    GB2312[398]:= 16#bef6;
    GB2312[399]:= 16#bff6;
    GB2312[400]:= 16#d2b1;
    GB2312[401]:= 16#c0e4;
    GB2312[402]:= 16#b6b3;
    GB2312[403]:= 16#d9fe;
    GB2312[404]:= 16#d9fd;
    GB2312[405]:= 16#bebb;
    GB2312[406]:= 16#c6e0;
    GB2312[407]:= 16#d7bc;
    GB2312[408]:= 16#daa1;
    GB2312[409]:= 16#c1b9;
    GB2312[410]:= 16#b5f2;
    GB2312[411]:= 16#c1e8;
    GB2312[412]:= 16#bcf5;
    GB2312[413]:= 16#b4d5;
    GB2312[414]:= 16#c1dd;
    GB2312[415]:= 16#c4fd;
    GB2312[416]:= 16#bcb8;
    GB2312[417]:= 16#b7b2;
    GB2312[418]:= 16#b7ef;
    GB2312[419]:= 16#d9ec;
    GB2312[420]:= 16#c6be;
    GB2312[421]:= 16#bfad;
    GB2312[422]:= 16#bbcb;
    GB2312[423]:= 16#b5ca;
    GB2312[424]:= 16#dbc9;
    GB2312[425]:= 16#d0d7;
    GB2312[426]:= 16#cdb9;
    GB2312[427]:= 16#b0bc;
    GB2312[428]:= 16#b3f6;
    GB2312[429]:= 16#bbf7;
    GB2312[430]:= 16#dbca;
    GB2312[431]:= 16#baaf;
    GB2312[432]:= 16#d4e4;
    GB2312[433]:= 16#b5b6;
    GB2312[434]:= 16#b5f3;
    GB2312[435]:= 16#d8d6;
    GB2312[436]:= 16#c8d0;
    GB2312[437]:= 16#b7d6;
    GB2312[438]:= 16#c7d0;
    GB2312[439]:= 16#d8d7;
    GB2312[440]:= 16#bfaf;
    GB2312[441]:= 16#dbbb;
    GB2312[442]:= 16#d8d8;
    GB2312[443]:= 16#d0cc;
    GB2312[444]:= 16#bbae;
    GB2312[445]:= 16#ebbe;
    GB2312[446]:= 16#c1d0;
    GB2312[447]:= 16#c1f5;
    GB2312[448]:= 16#d4f2;
    GB2312[449]:= 16#b8d5;
    GB2312[450]:= 16#b4b4;
    GB2312[451]:= 16#b3f5;
    GB2312[452]:= 16#c9be;
    GB2312[453]:= 16#c5d0;
    GB2312[454]:= 16#c5d9;
    GB2312[455]:= 16#c0fb;
    GB2312[456]:= 16#b1f0;
    GB2312[457]:= 16#d8d9;
    GB2312[458]:= 16#b9ce;
    GB2312[459]:= 16#b5bd;
    GB2312[460]:= 16#d8da;
    GB2312[461]:= 16#d6c6;
    GB2312[462]:= 16#cba2;
    GB2312[463]:= 16#c8af;
    GB2312[464]:= 16#c9b2;
    GB2312[465]:= 16#b4cc;
    GB2312[466]:= 16#bfcc;
    GB2312[467]:= 16#b9f4;
    GB2312[468]:= 16#d8db;
    GB2312[469]:= 16#d8dc;
    GB2312[470]:= 16#b6e7;
    GB2312[471]:= 16#bcc1;
    GB2312[472]:= 16#ccea;
    GB2312[473]:= 16#cff7;
    GB2312[474]:= 16#d8dd;
    GB2312[475]:= 16#c7b0;
    GB2312[476]:= 16#b9d0;
    GB2312[477]:= 16#bda3;
    GB2312[478]:= 16#ccde;
    GB2312[479]:= 16#c6ca;
    GB2312[480]:= 16#d8e0;
    GB2312[481]:= 16#d8de;
    GB2312[482]:= 16#d8df;
    GB2312[483]:= 16#b0fe;
    GB2312[484]:= 16#bee7;
    GB2312[485]:= 16#caa3;
    GB2312[486]:= 16#bcf4;
    GB2312[487]:= 16#b8b1;
    GB2312[488]:= 16#b8ee;
    GB2312[489]:= 16#d8e2;
    GB2312[490]:= 16#bdcb;
    GB2312[491]:= 16#d8e4;
    GB2312[492]:= 16#d8e3;
    GB2312[493]:= 16#c5fc;
    GB2312[494]:= 16#d8e5;
    GB2312[495]:= 16#d8e6;
    GB2312[496]:= 16#c1a6;
    GB2312[497]:= 16#c8b0;
    GB2312[498]:= 16#b0ec;
    GB2312[499]:= 16#b9a6;
    GB2312[500]:= 16#bcd3;
    GB2312[501]:= 16#cef1;
    GB2312[502]:= 16#dbbd;
    GB2312[503]:= 16#c1d3;
    GB2312[504]:= 16#b6af;
    GB2312[505]:= 16#d6fa;
    GB2312[506]:= 16#c5ac;
    GB2312[507]:= 16#bdd9;
    GB2312[508]:= 16#dbbe;
    GB2312[509]:= 16#dbbf;
    GB2312[510]:= 16#c0f8;
    GB2312[511]:= 16#bea2;
    GB2312[512]:= 16#c0cd;
    GB2312[513]:= 16#dbc0;
    GB2312[514]:= 16#cac6;
    GB2312[515]:= 16#b2aa;
    GB2312[516]:= 16#d3c2;
    GB2312[517]:= 16#c3e3;
    GB2312[518]:= 16#d1ab;
    GB2312[519]:= 16#dbc2;
    GB2312[520]:= 16#c0d5;
    GB2312[521]:= 16#dbc3;
    GB2312[522]:= 16#bfb1;
    GB2312[523]:= 16#c4bc;
    GB2312[524]:= 16#c7da;
    GB2312[525]:= 16#dbc4;
    GB2312[526]:= 16#d9e8;
    GB2312[527]:= 16#c9d7;
    GB2312[528]:= 16#b9b4;
    GB2312[529]:= 16#cef0;
    GB2312[530]:= 16#d4c8;
    GB2312[531]:= 16#b0fc;
    GB2312[532]:= 16#b4d2;
    GB2312[533]:= 16#d0d9;
    GB2312[534]:= 16#d9e9;
    GB2312[535]:= 16#decb;
    GB2312[536]:= 16#d9eb;
    GB2312[537]:= 16#d8b0;
    GB2312[538]:= 16#bbaf;
    GB2312[539]:= 16#b1b1;
    GB2312[540]:= 16#b3d7;
    GB2312[541]:= 16#d8ce;
    GB2312[542]:= 16#d4d1;
    GB2312[543]:= 16#bdb3;
    GB2312[544]:= 16#bfef;
    GB2312[545]:= 16#cfbb;
    GB2312[546]:= 16#d8d0;
    GB2312[547]:= 16#b7cb;
    GB2312[548]:= 16#d8d1;
    GB2312[549]:= 16#c6a5;
    GB2312[550]:= 16#c7f8;
    GB2312[551]:= 16#d2bd;
    GB2312[552]:= 16#d8d2;
    GB2312[553]:= 16#c4e4;
    GB2312[554]:= 16#caae;
    GB2312[555]:= 16#c7a7;
    GB2312[556]:= 16#d8a6;
    GB2312[557]:= 16#c9fd;
    GB2312[558]:= 16#cee7;
    GB2312[559]:= 16#bbdc;
    GB2312[560]:= 16#b0eb;
    GB2312[561]:= 16#bbaa;
    GB2312[562]:= 16#d0ad;
    GB2312[563]:= 16#b1b0;
    GB2312[564]:= 16#d7e4;
    GB2312[565]:= 16#d7bf;
    GB2312[566]:= 16#b5a5;
    GB2312[567]:= 16#c2f4;
    GB2312[568]:= 16#c4cf;
    GB2312[569]:= 16#b2a9;
    GB2312[570]:= 16#b2b7;
    GB2312[571]:= 16#b1e5;
    GB2312[572]:= 16#dfb2;
    GB2312[573]:= 16#d5bc;
    GB2312[574]:= 16#bfa8;
    GB2312[575]:= 16#c2ac;
    GB2312[576]:= 16#d8d5;
    GB2312[577]:= 16#c2b1;
    GB2312[578]:= 16#d8d4;
    GB2312[579]:= 16#ced4;
    GB2312[580]:= 16#dae0;
    GB2312[581]:= 16#cec0;
    GB2312[582]:= 16#d8b4;
    GB2312[583]:= 16#c3ae;
    GB2312[584]:= 16#d3a1;
    GB2312[585]:= 16#cea3;
    GB2312[586]:= 16#bcb4;
    GB2312[587]:= 16#c8b4;
    GB2312[588]:= 16#c2d1;
    GB2312[589]:= 16#beed;
    GB2312[590]:= 16#d0b6;
    GB2312[591]:= 16#dae1;
    GB2312[592]:= 16#c7e4;
    GB2312[593]:= 16#b3a7;
    GB2312[594]:= 16#b6f2;
    GB2312[595]:= 16#ccfc;
    GB2312[596]:= 16#c0fa;
    GB2312[597]:= 16#c0f7;
    GB2312[598]:= 16#d1b9;
    GB2312[599]:= 16#d1e1;
    GB2312[600]:= 16#d8c7;
    GB2312[601]:= 16#b2de;
    GB2312[602]:= 16#c0e5;
    GB2312[603]:= 16#baf1;
    GB2312[604]:= 16#d8c8;
    GB2312[605]:= 16#d4ad;
    GB2312[606]:= 16#cfe1;
    GB2312[607]:= 16#d8c9;
    GB2312[608]:= 16#d8ca;
    GB2312[609]:= 16#cfc3;
    GB2312[610]:= 16#b3f8;
    GB2312[611]:= 16#bec7;
    GB2312[612]:= 16#d8cb;
    GB2312[613]:= 16#dbcc;
    GB2312[614]:= 16#c8a5;
    GB2312[615]:= 16#cfd8;
    GB2312[616]:= 16#c8fe;
    GB2312[617]:= 16#b2ce;
    GB2312[618]:= 16#d3d6;
    GB2312[619]:= 16#b2e6;
    GB2312[620]:= 16#bcb0;
    GB2312[621]:= 16#d3d1;
    GB2312[622]:= 16#cbab;
    GB2312[623]:= 16#b7b4;
    GB2312[624]:= 16#b7a2;
    GB2312[625]:= 16#cae5;
    GB2312[626]:= 16#c8a1;
    GB2312[627]:= 16#cadc;
    GB2312[628]:= 16#b1e4;
    GB2312[629]:= 16#d0f0;
    GB2312[630]:= 16#c5d1;
    GB2312[631]:= 16#dbc5;
    GB2312[632]:= 16#b5fe;
    GB2312[633]:= 16#bfda;
    GB2312[634]:= 16#b9c5;
    GB2312[635]:= 16#bee4;
    GB2312[636]:= 16#c1ed;
    GB2312[637]:= 16#dfb6;
    GB2312[638]:= 16#dfb5;
    GB2312[639]:= 16#d6bb;
    GB2312[640]:= 16#bdd0;
    GB2312[641]:= 16#d5d9;
    GB2312[642]:= 16#b0c8;
    GB2312[643]:= 16#b6a3;
    GB2312[644]:= 16#bfc9;
    GB2312[645]:= 16#cca8;
    GB2312[646]:= 16#dfb3;
    GB2312[647]:= 16#cab7;
    GB2312[648]:= 16#d3d2;
    GB2312[649]:= 16#d8cf;
    GB2312[650]:= 16#d2b6;
    GB2312[651]:= 16#bac5;
    GB2312[652]:= 16#cbbe;
    GB2312[653]:= 16#ccbe;
    GB2312[654]:= 16#dfb7;
    GB2312[655]:= 16#b5f0;
    GB2312[656]:= 16#dfb4;
    GB2312[657]:= 16#d3f5;
    GB2312[658]:= 16#b3d4;
    GB2312[659]:= 16#b8f7;
    GB2312[660]:= 16#dfba;
    GB2312[661]:= 16#bacf;
    GB2312[662]:= 16#bcaa;
    GB2312[663]:= 16#b5f5;
    GB2312[664]:= 16#cdac;
    GB2312[665]:= 16#c3fb;
    GB2312[666]:= 16#baf3;
    GB2312[667]:= 16#c0f4;
    GB2312[668]:= 16#cdc2;
    GB2312[669]:= 16#cff2;
    GB2312[670]:= 16#dfb8;
    GB2312[671]:= 16#cfc5;
    GB2312[672]:= 16#c2c0;
    GB2312[673]:= 16#dfb9;
    GB2312[674]:= 16#c2f0;
    GB2312[675]:= 16#befd;
    GB2312[676]:= 16#c1df;
    GB2312[677]:= 16#cdcc;
    GB2312[678]:= 16#d2f7;
    GB2312[679]:= 16#b7cd;
    GB2312[680]:= 16#dfc1;
    GB2312[681]:= 16#dfc4;
    GB2312[682]:= 16#b7f1;
    GB2312[683]:= 16#b0c9;
    GB2312[684]:= 16#b6d6;
    GB2312[685]:= 16#b7d4;
    GB2312[686]:= 16#baac;
    GB2312[687]:= 16#ccfd;
    GB2312[688]:= 16#bfd4;
    GB2312[689]:= 16#cbb1;
    GB2312[690]:= 16#c6f4;
    GB2312[691]:= 16#d6a8;
    GB2312[692]:= 16#dfc5;
    GB2312[693]:= 16#cee2;
    GB2312[694]:= 16#b3b3;
    GB2312[695]:= 16#cefc;
    GB2312[696]:= 16#b4b5;
    GB2312[697]:= 16#cec7;
    GB2312[698]:= 16#baf0;
    GB2312[699]:= 16#cee1;
    GB2312[700]:= 16#d1bd;
    GB2312[701]:= 16#dfc0;
    GB2312[702]:= 16#b4f4;
    GB2312[703]:= 16#b3ca;
    GB2312[704]:= 16#b8e6;
    GB2312[705]:= 16#dfbb;
    GB2312[706]:= 16#c4c5;
    GB2312[707]:= 16#dfbc;
    GB2312[708]:= 16#dfbd;
    GB2312[709]:= 16#dfbe;
    GB2312[710]:= 16#c5bb;
    GB2312[711]:= 16#dfbf;
    GB2312[712]:= 16#dfc2;
    GB2312[713]:= 16#d4b1;
    GB2312[714]:= 16#dfc3;
    GB2312[715]:= 16#c7ba;
    GB2312[716]:= 16#ced8;
    GB2312[717]:= 16#c4d8;
    GB2312[718]:= 16#dfca;
    GB2312[719]:= 16#dfcf;
    GB2312[720]:= 16#d6dc;
    GB2312[721]:= 16#dfc9;
    GB2312[722]:= 16#dfda;
    GB2312[723]:= 16#ceb6;
    GB2312[724]:= 16#bac7;
    GB2312[725]:= 16#dfce;
    GB2312[726]:= 16#dfc8;
    GB2312[727]:= 16#c5de;
    GB2312[728]:= 16#c9eb;
    GB2312[729]:= 16#baf4;
    GB2312[730]:= 16#c3fc;
    GB2312[731]:= 16#bed7;
    GB2312[732]:= 16#dfc6;
    GB2312[733]:= 16#dfcd;
    GB2312[734]:= 16#c5d8;
    GB2312[735]:= 16#d5a6;
    GB2312[736]:= 16#bacd;
    GB2312[737]:= 16#becc;
    GB2312[738]:= 16#d3bd;
    GB2312[739]:= 16#b8c0;
    GB2312[740]:= 16#d6e4;
    GB2312[741]:= 16#dfc7;
    GB2312[742]:= 16#b9be;
    GB2312[743]:= 16#bfa7;
    GB2312[744]:= 16#c1fc;
    GB2312[745]:= 16#dfcb;
    GB2312[746]:= 16#dfcc;
    GB2312[747]:= 16#dfd0;
    GB2312[748]:= 16#dfdb;
    GB2312[749]:= 16#dfe5;
    GB2312[750]:= 16#dfd7;
    GB2312[751]:= 16#dfd6;
    GB2312[752]:= 16#d7c9;
    GB2312[753]:= 16#dfe3;
    GB2312[754]:= 16#dfe4;
    GB2312[755]:= 16#e5eb;
    GB2312[756]:= 16#d2a7;
    GB2312[757]:= 16#dfd2;
    GB2312[758]:= 16#bfa9;
    GB2312[759]:= 16#d4db;
    GB2312[760]:= 16#bfc8;
    GB2312[761]:= 16#dfd4;
    GB2312[762]:= 16#cfcc;
    GB2312[763]:= 16#dfdd;
    GB2312[764]:= 16#d1ca;
    GB2312[765]:= 16#dfde;
    GB2312[766]:= 16#b0a7;
    GB2312[767]:= 16#c6b7;
    GB2312[768]:= 16#dfd3;
    GB2312[769]:= 16#bae5;
    GB2312[770]:= 16#b6df;
    GB2312[771]:= 16#cddb;
    GB2312[772]:= 16#b9fe;
    GB2312[773]:= 16#d4d5;
    GB2312[774]:= 16#dfdf;
    GB2312[775]:= 16#cfec;
    GB2312[776]:= 16#b0a5;
    GB2312[777]:= 16#dfe7;
    GB2312[778]:= 16#dfd1;
    GB2312[779]:= 16#d1c6;
    GB2312[780]:= 16#dfd5;
    GB2312[781]:= 16#dfd8;
    GB2312[782]:= 16#dfd9;
    GB2312[783]:= 16#dfdc;
    GB2312[784]:= 16#bba9;
    GB2312[785]:= 16#dfe0;
    GB2312[786]:= 16#dfe1;
    GB2312[787]:= 16#dfe2;
    GB2312[788]:= 16#dfe6;
    GB2312[789]:= 16#dfe8;
    GB2312[790]:= 16#d3b4;
    GB2312[791]:= 16#b8e7;
    GB2312[792]:= 16#c5b6;
    GB2312[793]:= 16#dfea;
    GB2312[794]:= 16#c9da;
    GB2312[795]:= 16#c1a8;
    GB2312[796]:= 16#c4c4;
    GB2312[797]:= 16#bfde;
    GB2312[798]:= 16#cff8;
    GB2312[799]:= 16#d5dc;
    GB2312[800]:= 16#dfee;
    GB2312[801]:= 16#b2b8;
    GB2312[802]:= 16#badf;
    GB2312[803]:= 16#dfec;
    GB2312[804]:= 16#dbc1;
    GB2312[805]:= 16#d1e4;
    GB2312[806]:= 16#cbf4;
    GB2312[807]:= 16#b4bd;
    GB2312[808]:= 16#b0a6;
    GB2312[809]:= 16#dff1;
    GB2312[810]:= 16#ccc6;
    GB2312[811]:= 16#dff2;
    GB2312[812]:= 16#dfed;
    GB2312[813]:= 16#dfe9;
    GB2312[814]:= 16#dfeb;
    GB2312[815]:= 16#dfef;
    GB2312[816]:= 16#dff0;
    GB2312[817]:= 16#bbbd;
    GB2312[818]:= 16#dff3;
    GB2312[819]:= 16#dff4;
    GB2312[820]:= 16#bba3;
    GB2312[821]:= 16#cadb;
    GB2312[822]:= 16#cea8;
    GB2312[823]:= 16#e0a7;
    GB2312[824]:= 16#b3aa;
    GB2312[825]:= 16#e0a6;
    GB2312[826]:= 16#e0a1;
    GB2312[827]:= 16#dffe;
    GB2312[828]:= 16#cdd9;
    GB2312[829]:= 16#dffc;
    GB2312[830]:= 16#dffa;
    GB2312[831]:= 16#bfd0;
    GB2312[832]:= 16#d7c4;
    GB2312[833]:= 16#c9cc;
    GB2312[834]:= 16#dff8;
    GB2312[835]:= 16#b0a1;
    GB2312[836]:= 16#dffd;
    GB2312[837]:= 16#dffb;
    GB2312[838]:= 16#e0a2;
    GB2312[839]:= 16#e0a8;
    GB2312[840]:= 16#b7c8;
    GB2312[841]:= 16#c6a1;
    GB2312[842]:= 16#c9b6;
    GB2312[843]:= 16#c0b2;
    GB2312[844]:= 16#dff5;
    GB2312[845]:= 16#c5be;
    GB2312[846]:= 16#d8c4;
    GB2312[847]:= 16#dff9;
    GB2312[848]:= 16#c4f6;
    GB2312[849]:= 16#e0a3;
    GB2312[850]:= 16#e0a4;
    GB2312[851]:= 16#e0a5;
    GB2312[852]:= 16#d0a5;
    GB2312[853]:= 16#e0b4;
    GB2312[854]:= 16#cce4;
    GB2312[855]:= 16#e0b1;
    GB2312[856]:= 16#bfa6;
    GB2312[857]:= 16#e0af;
    GB2312[858]:= 16#ceb9;
    GB2312[859]:= 16#e0ab;
    GB2312[860]:= 16#c9c6;
    GB2312[861]:= 16#c0ae;
    GB2312[862]:= 16#e0ae;
    GB2312[863]:= 16#baed;
    GB2312[864]:= 16#bab0;
    GB2312[865]:= 16#e0a9;
    GB2312[866]:= 16#dff6;
    GB2312[867]:= 16#e0b3;
    GB2312[868]:= 16#e0b8;
    GB2312[869]:= 16#b4ad;
    GB2312[870]:= 16#e0b9;
    GB2312[871]:= 16#cfb2;
    GB2312[872]:= 16#bac8;
    GB2312[873]:= 16#e0b0;
    GB2312[874]:= 16#d0fa;
    GB2312[875]:= 16#e0ac;
    GB2312[876]:= 16#d4fb;
    GB2312[877]:= 16#dff7;
    GB2312[878]:= 16#c5e7;
    GB2312[879]:= 16#e0ad;
    GB2312[880]:= 16#d3f7;
    GB2312[881]:= 16#e0b6;
    GB2312[882]:= 16#e0b7;
    GB2312[883]:= 16#e0c4;
    GB2312[884]:= 16#d0e1;
    GB2312[885]:= 16#e0bc;
    GB2312[886]:= 16#e0c9;
    GB2312[887]:= 16#e0ca;
    GB2312[888]:= 16#e0be;
    GB2312[889]:= 16#e0aa;
    GB2312[890]:= 16#c9a4;
    GB2312[891]:= 16#e0c1;
    GB2312[892]:= 16#e0b2;
    GB2312[893]:= 16#cac8;
    GB2312[894]:= 16#e0c3;
    GB2312[895]:= 16#e0b5;
    GB2312[896]:= 16#cecb;
    GB2312[897]:= 16#cbc3;
    GB2312[898]:= 16#e0cd;
    GB2312[899]:= 16#e0c6;
    GB2312[900]:= 16#e0c2;
    GB2312[901]:= 16#e0cb;
    GB2312[902]:= 16#e0ba;
    GB2312[903]:= 16#e0bf;
    GB2312[904]:= 16#e0c0;
    GB2312[905]:= 16#e0c5;
    GB2312[906]:= 16#e0c7;
    GB2312[907]:= 16#e0c8;
    GB2312[908]:= 16#e0cc;
    GB2312[909]:= 16#e0bb;
    GB2312[910]:= 16#cbd4;
    GB2312[911]:= 16#e0d5;
    GB2312[912]:= 16#e0d6;
    GB2312[913]:= 16#e0d2;
    GB2312[914]:= 16#e0d0;
    GB2312[915]:= 16#bcce;
    GB2312[916]:= 16#e0d1;
    GB2312[917]:= 16#b8c2;
    GB2312[918]:= 16#d8c5;
    GB2312[919]:= 16#d0ea;
    GB2312[920]:= 16#c2ef;
    GB2312[921]:= 16#e0cf;
    GB2312[922]:= 16#e0bd;
    GB2312[923]:= 16#e0d4;
    GB2312[924]:= 16#e0d3;
    GB2312[925]:= 16#e0d7;
    GB2312[926]:= 16#e0dc;
    GB2312[927]:= 16#e0d8;
    GB2312[928]:= 16#d6f6;
    GB2312[929]:= 16#b3b0;
    GB2312[930]:= 16#d7ec;
    GB2312[931]:= 16#cbbb;
    GB2312[932]:= 16#e0da;
    GB2312[933]:= 16#cefb;
    GB2312[934]:= 16#bad9;
    GB2312[935]:= 16#e0e1;
    GB2312[936]:= 16#e0dd;
    GB2312[937]:= 16#d2ad;
    GB2312[938]:= 16#e0e2;
    GB2312[939]:= 16#e0db;
    GB2312[940]:= 16#e0d9;
    GB2312[941]:= 16#e0df;
    GB2312[942]:= 16#e0e0;
    GB2312[943]:= 16#e0de;
    GB2312[944]:= 16#e0e4;
    GB2312[945]:= 16#c6f7;
    GB2312[946]:= 16#d8ac;
    GB2312[947]:= 16#d4eb;
    GB2312[948]:= 16#e0e6;
    GB2312[949]:= 16#cac9;
    GB2312[950]:= 16#e0e5;
    GB2312[951]:= 16#b8c1;
    GB2312[952]:= 16#e0e7;
    GB2312[953]:= 16#e0e8;
    GB2312[954]:= 16#e0e9;
    GB2312[955]:= 16#e0e3;
    GB2312[956]:= 16#babf;
    GB2312[957]:= 16#cce7;
    GB2312[958]:= 16#e0ea;
    GB2312[959]:= 16#cff9;
    GB2312[960]:= 16#e0eb;
    GB2312[961]:= 16#c8c2;
    GB2312[962]:= 16#bdc0;
    GB2312[963]:= 16#c4d2;
    GB2312[964]:= 16#e0ec;
    GB2312[965]:= 16#e0ed;
    GB2312[966]:= 16#c7f4;
    GB2312[967]:= 16#cbc4;
    GB2312[968]:= 16#e0ee;
    GB2312[969]:= 16#bbd8;
    GB2312[970]:= 16#d8b6;
    GB2312[971]:= 16#d2f2;
    GB2312[972]:= 16#e0ef;
    GB2312[973]:= 16#cdc5;
    GB2312[974]:= 16#b6da;
    GB2312[975]:= 16#e0f1;
    GB2312[976]:= 16#d4b0;
    GB2312[977]:= 16#c0a7;
    GB2312[978]:= 16#b4d1;
    GB2312[979]:= 16#cea7;
    GB2312[980]:= 16#e0f0;
    GB2312[981]:= 16#e0f2;
    GB2312[982]:= 16#b9cc;
    GB2312[983]:= 16#b9fa;
    GB2312[984]:= 16#cdbc;
    GB2312[985]:= 16#e0f3;
    GB2312[986]:= 16#c6d4;
    GB2312[987]:= 16#e0f4;
    GB2312[988]:= 16#d4b2;
    GB2312[989]:= 16#c8a6;
    GB2312[990]:= 16#e0f6;
    GB2312[991]:= 16#e0f5;
    GB2312[992]:= 16#e0f7;
    GB2312[993]:= 16#cdc1;
    GB2312[994]:= 16#caa5;
    GB2312[995]:= 16#d4da;
    GB2312[996]:= 16#dbd7;
    GB2312[997]:= 16#dbd9;
    GB2312[998]:= 16#dbd8;
    GB2312[999]:= 16#b9e7;    //GB2312码 0000-999
END_IF;
(* Rung 12 *)
IF P_On THEN
    GB2312[1000]:= 16#dbdc;
    GB2312[1001]:= 16#dbdd;
    GB2312[1002]:= 16#b5d8;
    GB2312[1003]:= 16#dbda;
    GB2312[1004]:= 16#dbdb;
    GB2312[1005]:= 16#b3a1;
    GB2312[1006]:= 16#dbdf;
    GB2312[1007]:= 16#bbf8;
    GB2312[1008]:= 16#d6b7;
    GB2312[1009]:= 16#dbe0;
    GB2312[1010]:= 16#bef9;
    GB2312[1011]:= 16#b7bb;
    GB2312[1012]:= 16#dbd0;
    GB2312[1013]:= 16#ccae;
    GB2312[1014]:= 16#bfb2;
    GB2312[1015]:= 16#bbb5;
    GB2312[1016]:= 16#d7f8;
    GB2312[1017]:= 16#bfd3;
    GB2312[1018]:= 16#bfe9;
    GB2312[1019]:= 16#bce1;
    GB2312[1020]:= 16#ccb3;
    GB2312[1021]:= 16#dbde;
    GB2312[1022]:= 16#b0d3;
    GB2312[1023]:= 16#ceeb;
    GB2312[1024]:= 16#b7d8;
    GB2312[1025]:= 16#d7b9;
    GB2312[1026]:= 16#c6c2;
    GB2312[1027]:= 16#c0a4;
    GB2312[1028]:= 16#ccb9;
    GB2312[1029]:= 16#dbe7;
    GB2312[1030]:= 16#dbe1;
    GB2312[1031]:= 16#c6ba;
    GB2312[1032]:= 16#dbe3;
    GB2312[1033]:= 16#dbe8;
    GB2312[1034]:= 16#c5f7;
    GB2312[1035]:= 16#dbea;
    GB2312[1036]:= 16#dbe9;
    GB2312[1037]:= 16#bfc0;
    GB2312[1038]:= 16#dbe6;
    GB2312[1039]:= 16#dbe5;
    GB2312[1040]:= 16#b4b9;
    GB2312[1041]:= 16#c0ac;
    GB2312[1042]:= 16#c2a2;
    GB2312[1043]:= 16#dbe2;
    GB2312[1044]:= 16#dbe4;
    GB2312[1045]:= 16#d0cd;
    GB2312[1046]:= 16#dbed;
    GB2312[1047]:= 16#c0dd;
    GB2312[1048]:= 16#dbf2;
    GB2312[1049]:= 16#b6e2;
    GB2312[1050]:= 16#dbf3;
    GB2312[1051]:= 16#dbd2;
    GB2312[1052]:= 16#b9b8;
    GB2312[1053]:= 16#d4ab;
    GB2312[1054]:= 16#dbec;
    GB2312[1055]:= 16#bfd1;
    GB2312[1056]:= 16#dbf0;
    GB2312[1057]:= 16#dbd1;
    GB2312[1058]:= 16#b5e6;
    GB2312[1059]:= 16#dbeb;
    GB2312[1060]:= 16#bfe5;
    GB2312[1061]:= 16#dbee;
    GB2312[1062]:= 16#dbf1;
    GB2312[1063]:= 16#dbf9;
    GB2312[1064]:= 16#b9a1;
    GB2312[1065]:= 16#b0a3;
    GB2312[1066]:= 16#c2f1;
    GB2312[1067]:= 16#b3c7;
    GB2312[1068]:= 16#dbef;
    GB2312[1069]:= 16#dbf8;
    GB2312[1070]:= 16#c6d2;
    GB2312[1071]:= 16#dbf4;
    GB2312[1072]:= 16#dbf5;
    GB2312[1073]:= 16#dbf7;
    GB2312[1074]:= 16#dbf6;
    GB2312[1075]:= 16#dbfe;
    GB2312[1076]:= 16#d3f2;
    GB2312[1077]:= 16#b2ba;
    GB2312[1078]:= 16#dbfd;
    GB2312[1079]:= 16#dca4;
    GB2312[1080]:= 16#dbfb;
    GB2312[1081]:= 16#dbfa;
    GB2312[1082]:= 16#dbfc;
    GB2312[1083]:= 16#c5e0;
    GB2312[1084]:= 16#bbf9;
    GB2312[1085]:= 16#dca3;
    GB2312[1086]:= 16#dca5;
    GB2312[1087]:= 16#ccc3;
    GB2312[1088]:= 16#b6d1;
    GB2312[1089]:= 16#ddc0;
    GB2312[1090]:= 16#dca1;
    GB2312[1091]:= 16#dca2;
    GB2312[1092]:= 16#c7b5;
    GB2312[1093]:= 16#b6e9;
    GB2312[1094]:= 16#dca7;
    GB2312[1095]:= 16#dca6;
    GB2312[1096]:= 16#dca9;
    GB2312[1097]:= 16#b1a4;
    GB2312[1098]:= 16#b5cc;
    GB2312[1099]:= 16#bfb0;
    GB2312[1100]:= 16#d1df;
    GB2312[1101]:= 16#b6c2;
    GB2312[1102]:= 16#dca8;
    GB2312[1103]:= 16#cbfa;
    GB2312[1104]:= 16#ebf3;
    GB2312[1105]:= 16#cbdc;
    GB2312[1106]:= 16#cbfe;
    GB2312[1107]:= 16#ccc1;
    GB2312[1108]:= 16#c8fb;
    GB2312[1109]:= 16#dcaa;
    GB2312[1110]:= 16#ccee;
    GB2312[1111]:= 16#dcab;
    GB2312[1112]:= 16#dbd3;
    GB2312[1113]:= 16#dcaf;
    GB2312[1114]:= 16#dcac;
    GB2312[1115]:= 16#beb3;
    GB2312[1116]:= 16#cafb;
    GB2312[1117]:= 16#dcad;
    GB2312[1118]:= 16#c9ca;
    GB2312[1119]:= 16#c4b9;
    GB2312[1120]:= 16#c7bd;
    GB2312[1121]:= 16#dcae;
    GB2312[1122]:= 16#d4f6;
    GB2312[1123]:= 16#d0e6;
    GB2312[1124]:= 16#c4ab;
    GB2312[1125]:= 16#b6d5;
    GB2312[1126]:= 16#dbd4;
    GB2312[1127]:= 16#b1da;
    GB2312[1128]:= 16#dbd5;
    GB2312[1129]:= 16#dbd6;
    GB2312[1130]:= 16#babe;
    GB2312[1131]:= 16#c8c0;
    GB2312[1132]:= 16#cabf;
    GB2312[1133]:= 16#c8c9;
    GB2312[1134]:= 16#d7b3;
    GB2312[1135]:= 16#c9f9;
    GB2312[1136]:= 16#bfc7;
    GB2312[1137]:= 16#baf8;
    GB2312[1138]:= 16#d2bc;
    GB2312[1139]:= 16#e2ba;
    GB2312[1140]:= 16#b4a6;
    GB2312[1141]:= 16#b1b8;
    GB2312[1142]:= 16#b8b4;
    GB2312[1143]:= 16#cfc4;
    GB2312[1144]:= 16#d9e7;
    GB2312[1145]:= 16#cfa6;
    GB2312[1146]:= 16#cde2;
    GB2312[1147]:= 16#d9ed;
    GB2312[1148]:= 16#b6e0;
    GB2312[1149]:= 16#d2b9;
    GB2312[1150]:= 16#b9bb;
    GB2312[1151]:= 16#e2b9;
    GB2312[1152]:= 16#e2b7;
    GB2312[1153]:= 16#b4f3;
    GB2312[1154]:= 16#ccec;
    GB2312[1155]:= 16#ccab;
    GB2312[1156]:= 16#b7f2;
    GB2312[1157]:= 16#d8b2;
    GB2312[1158]:= 16#d1eb;
    GB2312[1159]:= 16#babb;
    GB2312[1160]:= 16#caa7;
    GB2312[1161]:= 16#cdb7;
    GB2312[1162]:= 16#d2c4;
    GB2312[1163]:= 16#bfe4;
    GB2312[1164]:= 16#bcd0;
    GB2312[1165]:= 16#b6e1;
    GB2312[1166]:= 16#dec5;
    GB2312[1167]:= 16#dec6;
    GB2312[1168]:= 16#dbbc;
    GB2312[1169]:= 16#d1d9;
    GB2312[1170]:= 16#c6e6;
    GB2312[1171]:= 16#c4ce;
    GB2312[1172]:= 16#b7ee;
    GB2312[1173]:= 16#b7dc;
    GB2312[1174]:= 16#bffc;
    GB2312[1175]:= 16#d7e0;
    GB2312[1176]:= 16#c6f5;
    GB2312[1177]:= 16#b1bc;
    GB2312[1178]:= 16#dec8;
    GB2312[1179]:= 16#bdb1;
    GB2312[1180]:= 16#ccd7;
    GB2312[1181]:= 16#deca;
    GB2312[1182]:= 16#dec9;
    GB2312[1183]:= 16#b5ec;
    GB2312[1184]:= 16#c9dd;
    GB2312[1185]:= 16#b0c2;
    GB2312[1186]:= 16#c5ae;
    GB2312[1187]:= 16#c5ab;
    GB2312[1188]:= 16#c4cc;
    GB2312[1189]:= 16#bce9;
    GB2312[1190]:= 16#cbfd;
    GB2312[1191]:= 16#bac3;
    GB2312[1192]:= 16#e5f9;
    GB2312[1193]:= 16#c8e7;
    GB2312[1194]:= 16#e5fa;
    GB2312[1195]:= 16#cdfd;
    GB2312[1196]:= 16#d7b1;
    GB2312[1197]:= 16#b8be;
    GB2312[1198]:= 16#c2e8;
    GB2312[1199]:= 16#c8d1;
    GB2312[1200]:= 16#e5fb;
    GB2312[1201]:= 16#b6ca;
    GB2312[1202]:= 16#bccb;
    GB2312[1203]:= 16#d1fd;
    GB2312[1204]:= 16#e6a1;
    GB2312[1205]:= 16#c3ee;
    GB2312[1206]:= 16#e6a4;
    GB2312[1207]:= 16#e5fe;
    GB2312[1208]:= 16#e6a5;
    GB2312[1209]:= 16#cdd7;
    GB2312[1210]:= 16#b7c1;
    GB2312[1211]:= 16#e5fc;
    GB2312[1212]:= 16#e5fd;
    GB2312[1213]:= 16#e6a3;
    GB2312[1214]:= 16#c4dd;
    GB2312[1215]:= 16#e6a8;
    GB2312[1216]:= 16#e6a7;
    GB2312[1217]:= 16#c3c3;
    GB2312[1218]:= 16#c6de;
    GB2312[1219]:= 16#e6aa;
    GB2312[1220]:= 16#c4b7;
    GB2312[1221]:= 16#e6a2;
    GB2312[1222]:= 16#cabc;
    GB2312[1223]:= 16#bde3;
    GB2312[1224]:= 16#b9c3;
    GB2312[1225]:= 16#e6a6;
    GB2312[1226]:= 16#d0d5;
    GB2312[1227]:= 16#ceaf;
    GB2312[1228]:= 16#e6a9;
    GB2312[1229]:= 16#e6b0;
    GB2312[1230]:= 16#d2a6;
    GB2312[1231]:= 16#bdaa;
    GB2312[1232]:= 16#e6ad;
    GB2312[1233]:= 16#e6af;
    GB2312[1234]:= 16#c0d1;
    GB2312[1235]:= 16#d2cc;
    GB2312[1236]:= 16#bca7;
    GB2312[1237]:= 16#e6b1;
    GB2312[1238]:= 16#d2f6;
    GB2312[1239]:= 16#d7cb;
    GB2312[1240]:= 16#cdfe;
    GB2312[1241]:= 16#cdde;
    GB2312[1242]:= 16#c2a6;
    GB2312[1243]:= 16#e6ab;
    GB2312[1244]:= 16#e6ac;
    GB2312[1245]:= 16#bdbf;
    GB2312[1246]:= 16#e6ae;
    GB2312[1247]:= 16#e6b3;
    GB2312[1248]:= 16#e6b2;
    GB2312[1249]:= 16#e6b6;
    GB2312[1250]:= 16#e6b8;
    GB2312[1251]:= 16#c4ef;
    GB2312[1252]:= 16#c4c8;
    GB2312[1253]:= 16#beea;
    GB2312[1254]:= 16#c9ef;
    GB2312[1255]:= 16#e6b7;
    GB2312[1256]:= 16#b6f0;
    GB2312[1257]:= 16#c3e4;
    GB2312[1258]:= 16#d3e9;
    GB2312[1259]:= 16#e6b4;
    GB2312[1260]:= 16#e6b5;
    GB2312[1261]:= 16#c8a2;
    GB2312[1262]:= 16#e6bd;
    GB2312[1263]:= 16#e6b9;
    GB2312[1264]:= 16#c6c5;
    GB2312[1265]:= 16#cdf1;
    GB2312[1266]:= 16#e6bb;
    GB2312[1267]:= 16#e6bc;
    GB2312[1268]:= 16#bbe9;
    GB2312[1269]:= 16#e6be;
    GB2312[1270]:= 16#e6ba;
    GB2312[1271]:= 16#c0b7;
    GB2312[1272]:= 16#d3a4;
    GB2312[1273]:= 16#e6bf;
    GB2312[1274]:= 16#c9f4;
    GB2312[1275]:= 16#e6c3;
    GB2312[1276]:= 16#e6c4;
    GB2312[1277]:= 16#d0f6;
    GB2312[1278]:= 16#c3bd;
    GB2312[1279]:= 16#c3c4;
    GB2312[1280]:= 16#e6c2;
    GB2312[1281]:= 16#e6c1;
    GB2312[1282]:= 16#e6c7;
    GB2312[1283]:= 16#cfb1;
    GB2312[1284]:= 16#ebf4;
    GB2312[1285]:= 16#e6ca;
    GB2312[1286]:= 16#e6c5;
    GB2312[1287]:= 16#bcde;
    GB2312[1288]:= 16#c9a9;
    GB2312[1289]:= 16#bcb5;
    GB2312[1290]:= 16#cfd3;
    GB2312[1291]:= 16#e6c8;
    GB2312[1292]:= 16#e6c9;
    GB2312[1293]:= 16#e6ce;
    GB2312[1294]:= 16#e6d0;
    GB2312[1295]:= 16#e6d1;
    GB2312[1296]:= 16#e6cb;
    GB2312[1297]:= 16#b5d5;
    GB2312[1298]:= 16#e6cc;
    GB2312[1299]:= 16#e6cf;
    GB2312[1300]:= 16#c4db;
    GB2312[1301]:= 16#e6c6;
    GB2312[1302]:= 16#e6cd;
    GB2312[1303]:= 16#e6d2;
    GB2312[1304]:= 16#e6d4;
    GB2312[1305]:= 16#e6d3;
    GB2312[1306]:= 16#e6d5;
    GB2312[1307]:= 16#d9f8;
    GB2312[1308]:= 16#e6d6;
    GB2312[1309]:= 16#e6d7;
    GB2312[1310]:= 16#d7d3;
    GB2312[1311]:= 16#e6dd;
    GB2312[1312]:= 16#e6de;
    GB2312[1313]:= 16#bfd7;
    GB2312[1314]:= 16#d4d0;
    GB2312[1315]:= 16#d7d6;
    GB2312[1316]:= 16#b4e6;
    GB2312[1317]:= 16#cbef;
    GB2312[1318]:= 16#e6da;
    GB2312[1319]:= 16#d8c3;
    GB2312[1320]:= 16#d7ce;
    GB2312[1321]:= 16#d0a2;
    GB2312[1322]:= 16#c3cf;
    GB2312[1323]:= 16#e6df;
    GB2312[1324]:= 16#bcbe;
    GB2312[1325]:= 16#b9c2;
    GB2312[1326]:= 16#e6db;
    GB2312[1327]:= 16#d1a7;
    GB2312[1328]:= 16#baa2;
    GB2312[1329]:= 16#c2cf;
    GB2312[1330]:= 16#d8ab;
    GB2312[1331]:= 16#caeb;
    GB2312[1332]:= 16#e5ee;
    GB2312[1333]:= 16#e6dc;
    GB2312[1334]:= 16#b7f5;
    GB2312[1335]:= 16#c8e6;
    GB2312[1336]:= 16#c4f5;
    GB2312[1337]:= 16#e5b2;
    GB2312[1338]:= 16#c4fe;
    GB2312[1339]:= 16#cbfc;
    GB2312[1340]:= 16#e5b3;
    GB2312[1341]:= 16#d5ac;
    GB2312[1342]:= 16#d3ee;
    GB2312[1343]:= 16#cad8;
    GB2312[1344]:= 16#b0b2;
    GB2312[1345]:= 16#cbce;
    GB2312[1346]:= 16#cdea;
    GB2312[1347]:= 16#baea;
    GB2312[1348]:= 16#e5b5;
    GB2312[1349]:= 16#e5b4;
    GB2312[1350]:= 16#d7da;
    GB2312[1351]:= 16#b9d9;
    GB2312[1352]:= 16#d6e6;
    GB2312[1353]:= 16#b6a8;
    GB2312[1354]:= 16#cdf0;
    GB2312[1355]:= 16#d2cb;
    GB2312[1356]:= 16#b1a6;
    GB2312[1357]:= 16#cab5;
    GB2312[1358]:= 16#b3e8;
    GB2312[1359]:= 16#c9f3;
    GB2312[1360]:= 16#bfcd;
    GB2312[1361]:= 16#d0fb;
    GB2312[1362]:= 16#cad2;
    GB2312[1363]:= 16#e5b6;
    GB2312[1364]:= 16#bbc2;
    GB2312[1365]:= 16#cfdc;
    GB2312[1366]:= 16#b9ac;
    GB2312[1367]:= 16#d4d7;
    GB2312[1368]:= 16#baa6;
    GB2312[1369]:= 16#d1e7;
    GB2312[1370]:= 16#cffc;
    GB2312[1371]:= 16#bcd2;
    GB2312[1372]:= 16#e5b7;
    GB2312[1373]:= 16#c8dd;
    GB2312[1374]:= 16#bfed;
    GB2312[1375]:= 16#b1f6;
    GB2312[1376]:= 16#cbde;
    GB2312[1377]:= 16#bcc5;
    GB2312[1378]:= 16#bcc4;
    GB2312[1379]:= 16#d2fa;
    GB2312[1380]:= 16#c3dc;
    GB2312[1381]:= 16#bfdc;
    GB2312[1382]:= 16#b8bb;
    GB2312[1383]:= 16#c3c2;
    GB2312[1384]:= 16#baae;
    GB2312[1385]:= 16#d4a2;
    GB2312[1386]:= 16#c7de;
    GB2312[1387]:= 16#c4af;
    GB2312[1388]:= 16#b2ec;
    GB2312[1389]:= 16#b9d1;
    GB2312[1390]:= 16#e5bb;
    GB2312[1391]:= 16#c1c8;
    GB2312[1392]:= 16#d5af;
    GB2312[1393]:= 16#e5bc;
    GB2312[1394]:= 16#e5be;
    GB2312[1395]:= 16#b4e7;
    GB2312[1396]:= 16#b6d4;
    GB2312[1397]:= 16#cbc2;
    GB2312[1398]:= 16#d1b0;
    GB2312[1399]:= 16#b5bc;
    GB2312[1400]:= 16#cad9;
    GB2312[1401]:= 16#b7e2;
    GB2312[1402]:= 16#c9e4;
    GB2312[1403]:= 16#bdab;
    GB2312[1404]:= 16#cebe;
    GB2312[1405]:= 16#d7f0;
    GB2312[1406]:= 16#d0a1;
    GB2312[1407]:= 16#c9d9;
    GB2312[1408]:= 16#b6fb;
    GB2312[1409]:= 16#e6d8;
    GB2312[1410]:= 16#bce2;
    GB2312[1411]:= 16#b3be;
    GB2312[1412]:= 16#c9d0;
    GB2312[1413]:= 16#e6d9;
    GB2312[1414]:= 16#b3a2;
    GB2312[1415]:= 16#decc;
    GB2312[1416]:= 16#d3c8;
    GB2312[1417]:= 16#decd;
    GB2312[1418]:= 16#d2a2;
    GB2312[1419]:= 16#dece;
    GB2312[1420]:= 16#becd;
    GB2312[1421]:= 16#decf;
    GB2312[1422]:= 16#caac;
    GB2312[1423]:= 16#d2fc;
    GB2312[1424]:= 16#b3df;
    GB2312[1425]:= 16#e5ea;
    GB2312[1426]:= 16#c4e1;
    GB2312[1427]:= 16#bea1;
    GB2312[1428]:= 16#ceb2;
    GB2312[1429]:= 16#c4f2;
    GB2312[1430]:= 16#bed6;
    GB2312[1431]:= 16#c6a8;
    GB2312[1432]:= 16#b2e3;
    GB2312[1433]:= 16#bed3;
    GB2312[1434]:= 16#c7fc;
    GB2312[1435]:= 16#cceb;
    GB2312[1436]:= 16#bdec;
    GB2312[1437]:= 16#cedd;
    GB2312[1438]:= 16#caba;
    GB2312[1439]:= 16#c6c1;
    GB2312[1440]:= 16#e5ec;
    GB2312[1441]:= 16#d0bc;
    GB2312[1442]:= 16#d5b9;
    GB2312[1443]:= 16#e5ed;
    GB2312[1444]:= 16#caf4;
    GB2312[1445]:= 16#cdc0;
    GB2312[1446]:= 16#c2c5;
    GB2312[1447]:= 16#e5ef;
    GB2312[1448]:= 16#c2c4;
    GB2312[1449]:= 16#e5f0;
    GB2312[1450]:= 16#e5f8;
    GB2312[1451]:= 16#cdcd;
    GB2312[1452]:= 16#c9bd;
    GB2312[1453]:= 16#d2d9;
    GB2312[1454]:= 16#e1a8;
    GB2312[1455]:= 16#d3ec;
    GB2312[1456]:= 16#cbea;
    GB2312[1457]:= 16#c6f1;
    GB2312[1458]:= 16#e1ac;
    GB2312[1459]:= 16#e1a7;
    GB2312[1460]:= 16#e1a9;
    GB2312[1461]:= 16#e1aa;
    GB2312[1462]:= 16#e1af;
    GB2312[1463]:= 16#b2ed;
    GB2312[1464]:= 16#e1ab;
    GB2312[1465]:= 16#b8da;
    GB2312[1466]:= 16#e1ad;
    GB2312[1467]:= 16#e1ae;
    GB2312[1468]:= 16#e1b0;
    GB2312[1469]:= 16#b5ba;
    GB2312[1470]:= 16#e1b1;
    GB2312[1471]:= 16#e1b3;
    GB2312[1472]:= 16#e1b8;
    GB2312[1473]:= 16#d1d2;
    GB2312[1474]:= 16#e1b6;
    GB2312[1475]:= 16#e1b5;
    GB2312[1476]:= 16#c1eb;
    GB2312[1477]:= 16#e1b7;
    GB2312[1478]:= 16#d4c0;
    GB2312[1479]:= 16#e1b2;
    GB2312[1480]:= 16#e1ba;
    GB2312[1481]:= 16#b0b6;
    GB2312[1482]:= 16#e1b4;
    GB2312[1483]:= 16#bff9;
    GB2312[1484]:= 16#e1b9;
    GB2312[1485]:= 16#e1bb;
    GB2312[1486]:= 16#e1be;
    GB2312[1487]:= 16#e1bc;
    GB2312[1488]:= 16#d6c5;
    GB2312[1489]:= 16#cfbf;
    GB2312[1490]:= 16#e1bd;
    GB2312[1491]:= 16#e1bf;
    GB2312[1492]:= 16#c2cd;
    GB2312[1493]:= 16#b6eb;
    GB2312[1494]:= 16#d3f8;
    GB2312[1495]:= 16#c7cd;
    GB2312[1496]:= 16#b7e5;
    GB2312[1497]:= 16#befe;
    GB2312[1498]:= 16#e1c0;
    GB2312[1499]:= 16#e1c1;
    GB2312[1500]:= 16#e1c7;
    GB2312[1501]:= 16#b3e7;
    GB2312[1502]:= 16#c6e9;
    GB2312[1503]:= 16#b4de;
    GB2312[1504]:= 16#d1c2;
    GB2312[1505]:= 16#e1c8;
    GB2312[1506]:= 16#e1c6;
    GB2312[1507]:= 16#e1c5;
    GB2312[1508]:= 16#e1c3;
    GB2312[1509]:= 16#e1c2;
    GB2312[1510]:= 16#b1c0;
    GB2312[1511]:= 16#d5b8;
    GB2312[1512]:= 16#e1c4;
    GB2312[1513]:= 16#e1cb;
    GB2312[1514]:= 16#e1cc;
    GB2312[1515]:= 16#e1ca;
    GB2312[1516]:= 16#effa;
    GB2312[1517]:= 16#e1d3;
    GB2312[1518]:= 16#e1d2;
    GB2312[1519]:= 16#c7b6;
    GB2312[1520]:= 16#e1c9;
    GB2312[1521]:= 16#e1ce;
    GB2312[1522]:= 16#e1d0;
    GB2312[1523]:= 16#e1d4;
    GB2312[1524]:= 16#e1d1;
    GB2312[1525]:= 16#e1cd;
    GB2312[1526]:= 16#e1cf;
    GB2312[1527]:= 16#e1d5;
    GB2312[1528]:= 16#e1d6;
    GB2312[1529]:= 16#e1d7;
    GB2312[1530]:= 16#e1d8;
    GB2312[1531]:= 16#e1da;
    GB2312[1532]:= 16#e1db;
    GB2312[1533]:= 16#cea1;
    GB2312[1534]:= 16#e7dd;
    GB2312[1535]:= 16#b4a8;
    GB2312[1536]:= 16#d6dd;
    GB2312[1537]:= 16#d1b2;
    GB2312[1538]:= 16#b3b2;
    GB2312[1539]:= 16#b9a4;
    GB2312[1540]:= 16#d7f3;
    GB2312[1541]:= 16#c7c9;
    GB2312[1542]:= 16#bede;
    GB2312[1543]:= 16#b9ae;
    GB2312[1544]:= 16#ced7;
    GB2312[1545]:= 16#b2ee;
    GB2312[1546]:= 16#dbcf;
    GB2312[1547]:= 16#bcba;
    GB2312[1548]:= 16#d2d1;
    GB2312[1549]:= 16#cbc8;
    GB2312[1550]:= 16#b0cd;
    GB2312[1551]:= 16#cfef;
    GB2312[1552]:= 16#d9e3;
    GB2312[1553]:= 16#bded;
    GB2312[1554]:= 16#b1d2;
    GB2312[1555]:= 16#cad0;
    GB2312[1556]:= 16#b2bc;
    GB2312[1557]:= 16#cba7;
    GB2312[1558]:= 16#b7ab;
    GB2312[1559]:= 16#caa6;
    GB2312[1560]:= 16#cfa3;
    GB2312[1561]:= 16#e0f8;
    GB2312[1562]:= 16#d5ca;
    GB2312[1563]:= 16#e0fb;
    GB2312[1564]:= 16#e0fa;
    GB2312[1565]:= 16#c5c1;
    GB2312[1566]:= 16#ccfb;
    GB2312[1567]:= 16#c1b1;
    GB2312[1568]:= 16#e0f9;
    GB2312[1569]:= 16#d6e3;
    GB2312[1570]:= 16#b2af;
    GB2312[1571]:= 16#d6c4;
    GB2312[1572]:= 16#b5db;
    GB2312[1573]:= 16#b4f8;
    GB2312[1574]:= 16#d6a1;
    GB2312[1575]:= 16#cfaf;
    GB2312[1576]:= 16#b0ef;
    GB2312[1577]:= 16#e0fc;
    GB2312[1578]:= 16#e1a1;
    GB2312[1579]:= 16#b3a3;
    GB2312[1580]:= 16#e0fd;
    GB2312[1581]:= 16#e0fe;
    GB2312[1582]:= 16#c3b1;
    GB2312[1583]:= 16#c3dd;
    GB2312[1584]:= 16#e1a2;
    GB2312[1585]:= 16#b7f9;
    GB2312[1586]:= 16#bbcf;
    GB2312[1587]:= 16#e1a3;
    GB2312[1588]:= 16#c4bb;
    GB2312[1589]:= 16#e1a4;
    GB2312[1590]:= 16#e1a5;
    GB2312[1591]:= 16#e1a6;
    GB2312[1592]:= 16#b4b1;
    GB2312[1593]:= 16#b8c9;
    GB2312[1594]:= 16#c6bd;
    GB2312[1595]:= 16#c4ea;
    GB2312[1596]:= 16#b2a2;
    GB2312[1597]:= 16#d0d2;
    GB2312[1598]:= 16#e7db;
    GB2312[1599]:= 16#bbc3;
    GB2312[1600]:= 16#d3d7;
    GB2312[1601]:= 16#d3c4;
    GB2312[1602]:= 16#b9e3;
    GB2312[1603]:= 16#e2cf;
    GB2312[1604]:= 16#d7af;
    GB2312[1605]:= 16#c7ec;
    GB2312[1606]:= 16#b1d3;
    GB2312[1607]:= 16#b4b2;
    GB2312[1608]:= 16#e2d1;
    GB2312[1609]:= 16#d0f2;
    GB2312[1610]:= 16#c2ae;
    GB2312[1611]:= 16#e2d0;
    GB2312[1612]:= 16#bfe2;
    GB2312[1613]:= 16#d3a6;
    GB2312[1614]:= 16#b5d7;
    GB2312[1615]:= 16#e2d2;
    GB2312[1616]:= 16#b5ea;
    GB2312[1617]:= 16#c3ed;
    GB2312[1618]:= 16#b8fd;
    GB2312[1619]:= 16#b8ae;
    GB2312[1620]:= 16#c5d3;
    GB2312[1621]:= 16#b7cf;
    GB2312[1622]:= 16#e2d4;
    GB2312[1623]:= 16#e2d3;
    GB2312[1624]:= 16#b6c8;
    GB2312[1625]:= 16#d7f9;
    GB2312[1626]:= 16#cda5;
    GB2312[1627]:= 16#e2d8;
    GB2312[1628]:= 16#e2d6;
    GB2312[1629]:= 16#cafc;
    GB2312[1630]:= 16#bfb5;
    GB2312[1631]:= 16#d3b9;
    GB2312[1632]:= 16#e2d5;
    GB2312[1633]:= 16#e2d7;
    GB2312[1634]:= 16#c1ae;
    GB2312[1635]:= 16#c0c8;
    GB2312[1636]:= 16#e2db;
    GB2312[1637]:= 16#e2da;
    GB2312[1638]:= 16#c0aa;
    GB2312[1639]:= 16#c1ce;
    GB2312[1640]:= 16#e2dc;
    GB2312[1641]:= 16#e2dd;
    GB2312[1642]:= 16#e2de;
    GB2312[1643]:= 16#dbc8;
    GB2312[1644]:= 16#d1d3;
    GB2312[1645]:= 16#cda2;
    GB2312[1646]:= 16#bda8;
    GB2312[1647]:= 16#dec3;
    GB2312[1648]:= 16#d8a5;
    GB2312[1649]:= 16#bfaa;
    GB2312[1650]:= 16#dbcd;
    GB2312[1651]:= 16#d2ec;
    GB2312[1652]:= 16#c6fa;
    GB2312[1653]:= 16#c5aa;
    GB2312[1654]:= 16#dec4;
    GB2312[1655]:= 16#b1d7;
    GB2312[1656]:= 16#dfae;
    GB2312[1657]:= 16#cabd;
    GB2312[1658]:= 16#dfb1;
    GB2312[1659]:= 16#b9ad;
    GB2312[1660]:= 16#d2fd;
    GB2312[1661]:= 16#b8a5;
    GB2312[1662]:= 16#baeb;
    GB2312[1663]:= 16#b3da;
    GB2312[1664]:= 16#b5dc;
    GB2312[1665]:= 16#d5c5;
    GB2312[1666]:= 16#c3d6;
    GB2312[1667]:= 16#cfd2;
    GB2312[1668]:= 16#bba1;
    GB2312[1669]:= 16#e5f3;
    GB2312[1670]:= 16#e5f2;
    GB2312[1671]:= 16#e5f4;
    GB2312[1672]:= 16#cde4;
    GB2312[1673]:= 16#c8f5;
    GB2312[1674]:= 16#b5af;
    GB2312[1675]:= 16#c7bf;
    GB2312[1676]:= 16#e5f6;
    GB2312[1677]:= 16#ecb0;
    GB2312[1678]:= 16#e5e6;
    GB2312[1679]:= 16#b9e9;
    GB2312[1680]:= 16#b5b1;
    GB2312[1681]:= 16#c2bc;
    GB2312[1682]:= 16#e5e8;
    GB2312[1683]:= 16#e5e7;
    GB2312[1684]:= 16#e5e9;
    GB2312[1685]:= 16#d2cd;
    GB2312[1686]:= 16#e1ea;
    GB2312[1687]:= 16#d0ce;
    GB2312[1688]:= 16#cdae;
    GB2312[1689]:= 16#d1e5;
    GB2312[1690]:= 16#b2ca;
    GB2312[1691]:= 16#b1eb;
    GB2312[1692]:= 16#b1f2;
    GB2312[1693]:= 16#c5ed;
    GB2312[1694]:= 16#d5c3;
    GB2312[1695]:= 16#d3b0;
    GB2312[1696]:= 16#e1dc;
    GB2312[1697]:= 16#e1dd;
    GB2312[1698]:= 16#d2db;
    GB2312[1699]:= 16#b3b9;
    GB2312[1700]:= 16#b1cb;
    GB2312[1701]:= 16#cdf9;
    GB2312[1702]:= 16#d5f7;
    GB2312[1703]:= 16#e1de;
    GB2312[1704]:= 16#beb6;
    GB2312[1705]:= 16#b4fd;
    GB2312[1706]:= 16#e1df;
    GB2312[1707]:= 16#badc;
    GB2312[1708]:= 16#e1e0;
    GB2312[1709]:= 16#bbb2;
    GB2312[1710]:= 16#c2c9;
    GB2312[1711]:= 16#e1e1;
    GB2312[1712]:= 16#d0ec;
    GB2312[1713]:= 16#cdbd;
    GB2312[1714]:= 16#e1e2;
    GB2312[1715]:= 16#b5c3;
    GB2312[1716]:= 16#c5c7;
    GB2312[1717]:= 16#e1e3;
    GB2312[1718]:= 16#e1e4;
    GB2312[1719]:= 16#d3f9;
    GB2312[1720]:= 16#e1e5;
    GB2312[1721]:= 16#d1ad;
    GB2312[1722]:= 16#e1e6;
    GB2312[1723]:= 16#cea2;
    GB2312[1724]:= 16#e1e7;
    GB2312[1725]:= 16#b5c2;
    GB2312[1726]:= 16#e1e8;
    GB2312[1727]:= 16#bbd5;
    GB2312[1728]:= 16#d0c4;
    GB2312[1729]:= 16#e2e0;
    GB2312[1730]:= 16#b1d8;
    GB2312[1731]:= 16#d2e4;
    GB2312[1732]:= 16#e2e1;
    GB2312[1733]:= 16#bcc9;
    GB2312[1734]:= 16#c8cc;
    GB2312[1735]:= 16#e2e3;
    GB2312[1736]:= 16#ecfe;
    GB2312[1737]:= 16#ecfd;
    GB2312[1738]:= 16#dfaf;
    GB2312[1739]:= 16#e2e2;
    GB2312[1740]:= 16#d6be;
    GB2312[1741]:= 16#cdfc;
    GB2312[1742]:= 16#c3a6;
    GB2312[1743]:= 16#e3c3;
    GB2312[1744]:= 16#d6d2;
    GB2312[1745]:= 16#e2e7;
    GB2312[1746]:= 16#e2e8;
    GB2312[1747]:= 16#d3c7;
    GB2312[1748]:= 16#e2ec;
    GB2312[1749]:= 16#bfec;
    GB2312[1750]:= 16#e2ed;
    GB2312[1751]:= 16#e2e5;
    GB2312[1752]:= 16#b3c0;
    GB2312[1753]:= 16#c4ee;
    GB2312[1754]:= 16#e2ee;
    GB2312[1755]:= 16#d0c3;
    GB2312[1756]:= 16#baf6;
    GB2312[1757]:= 16#e2e9;
    GB2312[1758]:= 16#b7de;
    GB2312[1759]:= 16#bbb3;
    GB2312[1760]:= 16#ccac;
    GB2312[1761]:= 16#cbcb;
    GB2312[1762]:= 16#e2e4;
    GB2312[1763]:= 16#e2e6;
    GB2312[1764]:= 16#e2ea;
    GB2312[1765]:= 16#e2eb;
    GB2312[1766]:= 16#e2f7;
    GB2312[1767]:= 16#e2f4;
    GB2312[1768]:= 16#d4f5;
    GB2312[1769]:= 16#e2f3;
    GB2312[1770]:= 16#c5ad;
    GB2312[1771]:= 16#d5fa;
    GB2312[1772]:= 16#c5c2;
    GB2312[1773]:= 16#b2c0;
    GB2312[1774]:= 16#e2ef;
    GB2312[1775]:= 16#e2f2;
    GB2312[1776]:= 16#c1af;
    GB2312[1777]:= 16#cbbc;
    GB2312[1778]:= 16#b5a1;
    GB2312[1779]:= 16#e2f9;
    GB2312[1780]:= 16#bcb1;
    GB2312[1781]:= 16#e2f1;
    GB2312[1782]:= 16#d0d4;
    GB2312[1783]:= 16#d4b9;
    GB2312[1784]:= 16#e2f5;
    GB2312[1785]:= 16#b9d6;
    GB2312[1786]:= 16#e2f6;
    GB2312[1787]:= 16#c7d3;
    GB2312[1788]:= 16#e2f0;
    GB2312[1789]:= 16#d7dc;
    GB2312[1790]:= 16#eda1;
    GB2312[1791]:= 16#e2f8;
    GB2312[1792]:= 16#eda5;
    GB2312[1793]:= 16#e2fe;
    GB2312[1794]:= 16#cad1;
    GB2312[1795]:= 16#c1b5;
    GB2312[1796]:= 16#bbd0;
    GB2312[1797]:= 16#bfd6;
    GB2312[1798]:= 16#bae3;
    GB2312[1799]:= 16#cba1;
    GB2312[1800]:= 16#eda6;
    GB2312[1801]:= 16#eda3;
    GB2312[1802]:= 16#eda2;
    GB2312[1803]:= 16#bbd6;
    GB2312[1804]:= 16#eda7;
    GB2312[1805]:= 16#d0f4;
    GB2312[1806]:= 16#eda4;
    GB2312[1807]:= 16#bade;
    GB2312[1808]:= 16#b6f7;
    GB2312[1809]:= 16#e3a1;
    GB2312[1810]:= 16#b6b2;
    GB2312[1811]:= 16#ccf1;
    GB2312[1812]:= 16#b9a7;
    GB2312[1813]:= 16#cfa2;
    GB2312[1814]:= 16#c7a1;
    GB2312[1815]:= 16#bfd2;
    GB2312[1816]:= 16#b6f1;
    GB2312[1817]:= 16#e2fa;
    GB2312[1818]:= 16#e2fb;
    GB2312[1819]:= 16#e2fd;
    GB2312[1820]:= 16#e2fc;
    GB2312[1821]:= 16#c4d5;
    GB2312[1822]:= 16#e3a2;
    GB2312[1823]:= 16#d3c1;
    GB2312[1824]:= 16#e3a7;
    GB2312[1825]:= 16#c7c4;
    GB2312[1826]:= 16#cfa4;
    GB2312[1827]:= 16#e3a9;
    GB2312[1828]:= 16#bab7;
    GB2312[1829]:= 16#e3a8;
    GB2312[1830]:= 16#bbda;
    GB2312[1831]:= 16#e3a3;
    GB2312[1832]:= 16#e3a4;
    GB2312[1833]:= 16#e3aa;
    GB2312[1834]:= 16#e3a6;
    GB2312[1835]:= 16#cef2;
    GB2312[1836]:= 16#d3c6;
    GB2312[1837]:= 16#bbbc;
    GB2312[1838]:= 16#d4c3;
    GB2312[1839]:= 16#c4fa;
    GB2312[1840]:= 16#eda8;
    GB2312[1841]:= 16#d0fc;
    GB2312[1842]:= 16#e3a5;
    GB2312[1843]:= 16#c3f5;
    GB2312[1844]:= 16#e3ad;
    GB2312[1845]:= 16#b1af;
    GB2312[1846]:= 16#e3b2;
    GB2312[1847]:= 16#bcc2;
    GB2312[1848]:= 16#e3ac;
    GB2312[1849]:= 16#b5bf;
    GB2312[1850]:= 16#c7e9;
    GB2312[1851]:= 16#e3b0;
    GB2312[1852]:= 16#beaa;
    GB2312[1853]:= 16#cdef;
    GB2312[1854]:= 16#bbf3;
    GB2312[1855]:= 16#cce8;
    GB2312[1856]:= 16#e3af;
    GB2312[1857]:= 16#e3b1;
    GB2312[1858]:= 16#cfa7;
    GB2312[1859]:= 16#e3ae;
    GB2312[1860]:= 16#cea9;
    GB2312[1861]:= 16#bbdd;
    GB2312[1862]:= 16#b5eb;
    GB2312[1863]:= 16#bee5;
    GB2312[1864]:= 16#b2d2;
    GB2312[1865]:= 16#b3cd;
    GB2312[1866]:= 16#b1b9;
    GB2312[1867]:= 16#e3ab;
    GB2312[1868]:= 16#b2d1;
    GB2312[1869]:= 16#b5ac;
    GB2312[1870]:= 16#b9df;
    GB2312[1871]:= 16#b6e8;
    GB2312[1872]:= 16#cfeb;
    GB2312[1873]:= 16#e3b7;
    GB2312[1874]:= 16#bbcc;
    GB2312[1875]:= 16#c8c7;
    GB2312[1876]:= 16#d0ca;
    GB2312[1877]:= 16#e3b8;
    GB2312[1878]:= 16#b3ee;
    GB2312[1879]:= 16#eda9;
    GB2312[1880]:= 16#d3fa;
    GB2312[1881]:= 16#d3e4;
    GB2312[1882]:= 16#edaa;
    GB2312[1883]:= 16#e3b9;
    GB2312[1884]:= 16#d2e2;
    GB2312[1885]:= 16#e3b5;
    GB2312[1886]:= 16#d3de;
    GB2312[1887]:= 16#b8d0;
    GB2312[1888]:= 16#e3b3;
    GB2312[1889]:= 16#e3b6;
    GB2312[1890]:= 16#b7df;
    GB2312[1891]:= 16#e3b4;
    GB2312[1892]:= 16#c0a2;
    GB2312[1893]:= 16#e3ba;
    GB2312[1894]:= 16#d4b8;
    GB2312[1895]:= 16#b4c8;
    GB2312[1896]:= 16#e3bb;
    GB2312[1897]:= 16#bbc5;
    GB2312[1898]:= 16#c9f7;
    GB2312[1899]:= 16#c9e5;
    GB2312[1900]:= 16#c4bd;
    GB2312[1901]:= 16#edab;
    GB2312[1902]:= 16#c2fd;
    GB2312[1903]:= 16#bbdb;
    GB2312[1904]:= 16#bfae;
    GB2312[1905]:= 16#cebf;
    GB2312[1906]:= 16#e3bc;
    GB2312[1907]:= 16#bfb6;
    GB2312[1908]:= 16#b1ef;
    GB2312[1909]:= 16#d4f7;
    GB2312[1910]:= 16#e3be;
    GB2312[1911]:= 16#edad;
    GB2312[1912]:= 16#e3bf;
    GB2312[1913]:= 16#baa9;
    GB2312[1914]:= 16#edac;
    GB2312[1915]:= 16#e3bd;
    GB2312[1916]:= 16#e3c0;
    GB2312[1917]:= 16#bab6;
    GB2312[1918]:= 16#b6ae;
    GB2312[1919]:= 16#d0b8;
    GB2312[1920]:= 16#b0c3;
    GB2312[1921]:= 16#edae;
    GB2312[1922]:= 16#edaf;
    GB2312[1923]:= 16#c0c1;
    GB2312[1924]:= 16#e3c1;
    GB2312[1925]:= 16#c5b3;
    GB2312[1926]:= 16#e3c2;
    GB2312[1927]:= 16#dcb2;
    GB2312[1928]:= 16#edb0;
    GB2312[1929]:= 16#b8ea;
    GB2312[1930]:= 16#ceec;
    GB2312[1931]:= 16#eaa7;
    GB2312[1932]:= 16#d0e7;
    GB2312[1933]:= 16#caf9;
    GB2312[1934]:= 16#c8d6;
    GB2312[1935]:= 16#cfb7;
    GB2312[1936]:= 16#b3c9;
    GB2312[1937]:= 16#ced2;
    GB2312[1938]:= 16#bde4;
    GB2312[1939]:= 16#e3de;
    GB2312[1940]:= 16#bbf2;
    GB2312[1941]:= 16#eaa8;
    GB2312[1942]:= 16#d5bd;
    GB2312[1943]:= 16#c6dd;
    GB2312[1944]:= 16#eaa9;
    GB2312[1945]:= 16#eaaa;
    GB2312[1946]:= 16#eaac;
    GB2312[1947]:= 16#eaab;
    GB2312[1948]:= 16#eaae;
    GB2312[1949]:= 16#eaad;
    GB2312[1950]:= 16#bdd8;
    GB2312[1951]:= 16#eaaf;
    GB2312[1952]:= 16#c2be;
    GB2312[1953]:= 16#b4c1;
    GB2312[1954]:= 16#b4f7;
    GB2312[1955]:= 16#bba7;
    GB2312[1956]:= 16#ece6;
    GB2312[1957]:= 16#ece5;
    GB2312[1958]:= 16#b7bf;
    GB2312[1959]:= 16#cbf9;
    GB2312[1960]:= 16#b1e2;
    GB2312[1961]:= 16#ece7;
    GB2312[1962]:= 16#c9c8;
    GB2312[1963]:= 16#ece8;
    GB2312[1964]:= 16#ece9;
    GB2312[1965]:= 16#cad6;
    GB2312[1966]:= 16#ded0;
    GB2312[1967]:= 16#b2c5;
    GB2312[1968]:= 16#d4fa;
    GB2312[1969]:= 16#c6cb;
    GB2312[1970]:= 16#b0c7;
    GB2312[1971]:= 16#b4f2;
    GB2312[1972]:= 16#c8d3;
    GB2312[1973]:= 16#cdd0;
    GB2312[1974]:= 16#bfb8;
    GB2312[1975]:= 16#bfdb;
    GB2312[1976]:= 16#c7a4;
    GB2312[1977]:= 16#d6b4;
    GB2312[1978]:= 16#c0a9;
    GB2312[1979]:= 16#ded1;
    GB2312[1980]:= 16#c9a8;
    GB2312[1981]:= 16#d1ef;
    GB2312[1982]:= 16#c5a4;
    GB2312[1983]:= 16#b0e7;
    GB2312[1984]:= 16#b3b6;
    GB2312[1985]:= 16#c8c5;
    GB2312[1986]:= 16#b0e2;
    GB2312[1987]:= 16#b7f6;
    GB2312[1988]:= 16#c5fa;
    GB2312[1989]:= 16#b6f3;
    GB2312[1990]:= 16#d5d2;
    GB2312[1991]:= 16#b3d0;
    GB2312[1992]:= 16#bcbc;
    GB2312[1993]:= 16#b3ad;
    GB2312[1994]:= 16#bef1;
    GB2312[1995]:= 16#b0d1;
    GB2312[1996]:= 16#d2d6;
    GB2312[1997]:= 16#cae3;
    GB2312[1998]:= 16#d7a5;
    GB2312[1999]:= 16#cdb6;    //GB2312码 1000-1999
END_IF;

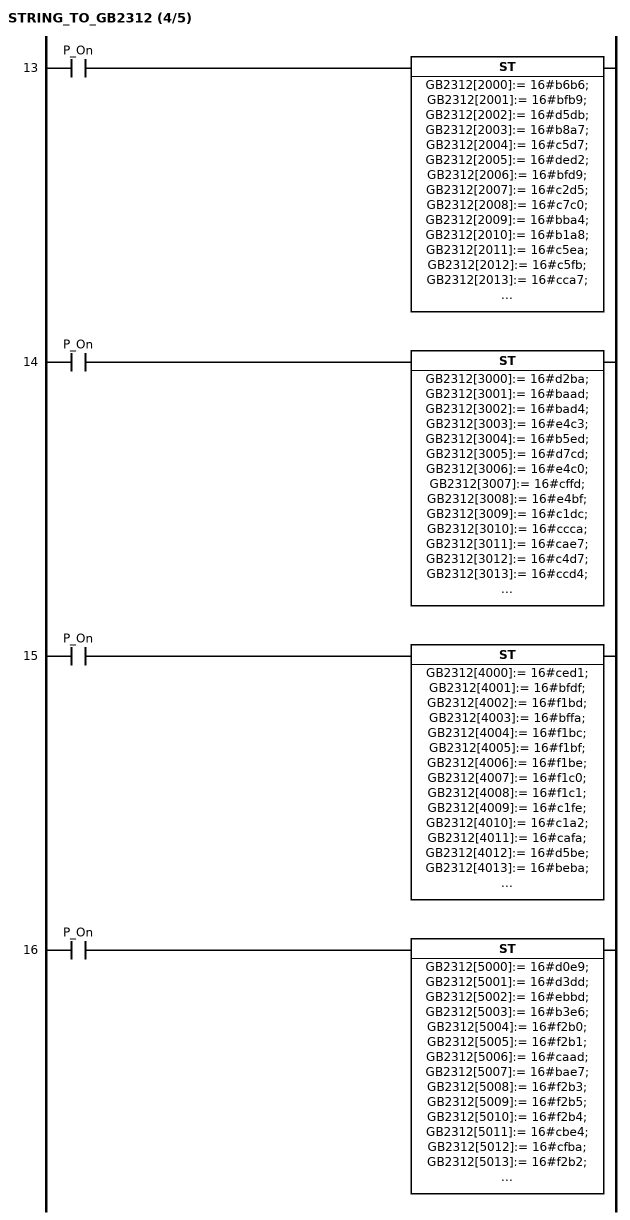
(* [picture p4: STRING_TO_GB2312, rungs 13-16] *)
(* Rung 13 *)
IF P_On THEN
    GB2312[2000]:= 16#b6b6;
    GB2312[2001]:= 16#bfb9;
    GB2312[2002]:= 16#d5db;
    GB2312[2003]:= 16#b8a7;
    GB2312[2004]:= 16#c5d7;
    GB2312[2005]:= 16#ded2;
    GB2312[2006]:= 16#bfd9;
    GB2312[2007]:= 16#c2d5;
    GB2312[2008]:= 16#c7c0;
    GB2312[2009]:= 16#bba4;
    GB2312[2010]:= 16#b1a8;
    GB2312[2011]:= 16#c5ea;
    GB2312[2012]:= 16#c5fb;
    GB2312[2013]:= 16#cca7;
    GB2312[2014]:= 16#b1a7;
    GB2312[2015]:= 16#b5d6;
    GB2312[2016]:= 16#c4a8;
    GB2312[2017]:= 16#ded3;
    GB2312[2018]:= 16#d1ba;
    GB2312[2019]:= 16#b3e9;
    GB2312[2020]:= 16#c3f2;
    GB2312[2021]:= 16#b7f7;
    GB2312[2022]:= 16#d6f4;
    GB2312[2023]:= 16#b5a3;
    GB2312[2024]:= 16#b2f0;
    GB2312[2025]:= 16#c4b4;
    GB2312[2026]:= 16#c4e9;
    GB2312[2027]:= 16#c0ad;
    GB2312[2028]:= 16#ded4;
    GB2312[2029]:= 16#b0e8;
    GB2312[2030]:= 16#c5c4;
    GB2312[2031]:= 16#c1e0;
    GB2312[2032]:= 16#b9d5;
    GB2312[2033]:= 16#bedc;
    GB2312[2034]:= 16#cdd8;
    GB2312[2035]:= 16#b0ce;
    GB2312[2036]:= 16#cdcf;
    GB2312[2037]:= 16#ded6;
    GB2312[2038]:= 16#bed0;
    GB2312[2039]:= 16#d7be;
    GB2312[2040]:= 16#ded5;
    GB2312[2041]:= 16#d5d0;
    GB2312[2042]:= 16#b0dd;
    GB2312[2043]:= 16#c4e2;
    GB2312[2044]:= 16#c2a3;
    GB2312[2045]:= 16#bcf0;
    GB2312[2046]:= 16#d3b5;
    GB2312[2047]:= 16#c0b9;
    GB2312[2048]:= 16#c5a1;
    GB2312[2049]:= 16#b2a6;
    GB2312[2050]:= 16#d4f1;
    GB2312[2051]:= 16#c0a8;
    GB2312[2052]:= 16#cac3;
    GB2312[2053]:= 16#ded7;
    GB2312[2054]:= 16#d5fc;
    GB2312[2055]:= 16#b9b0;
    GB2312[2056]:= 16#c8ad;
    GB2312[2057]:= 16#cba9;
    GB2312[2058]:= 16#ded9;
    GB2312[2059]:= 16#bfbd;
    GB2312[2060]:= 16#c6b4;
    GB2312[2061]:= 16#d7a7;
    GB2312[2062]:= 16#cab0;
    GB2312[2063]:= 16#c4c3;
    GB2312[2064]:= 16#b3d6;
    GB2312[2065]:= 16#b9d2;
    GB2312[2066]:= 16#d6b8;
    GB2312[2067]:= 16#eafc;
    GB2312[2068]:= 16#b0b4;
    GB2312[2069]:= 16#bfe6;
    GB2312[2070]:= 16#ccf4;
    GB2312[2071]:= 16#cdda;
    GB2312[2072]:= 16#d6bf;
    GB2312[2073]:= 16#c2ce;
    GB2312[2074]:= 16#cece;
    GB2312[2075]:= 16#cca2;
    GB2312[2076]:= 16#d0ae;
    GB2312[2077]:= 16#c4d3;
    GB2312[2078]:= 16#b5b2;
    GB2312[2079]:= 16#ded8;
    GB2312[2080]:= 16#d5f5;
    GB2312[2081]:= 16#bcb7;
    GB2312[2082]:= 16#bbd3;
    GB2312[2083]:= 16#b0a4;
    GB2312[2084]:= 16#c5b2;
    GB2312[2085]:= 16#b4ec;
    GB2312[2086]:= 16#d5f1;
    GB2312[2087]:= 16#eafd;
    GB2312[2088]:= 16#deda;
    GB2312[2089]:= 16#cda6;
    GB2312[2090]:= 16#cdec;
    GB2312[2091]:= 16#cee6;
    GB2312[2092]:= 16#dedc;
    GB2312[2093]:= 16#cdb1;
    GB2312[2094]:= 16#c0a6;
    GB2312[2095]:= 16#d7bd;
    GB2312[2096]:= 16#dedb;
    GB2312[2097]:= 16#b0c6;
    GB2312[2098]:= 16#bab4;
    GB2312[2099]:= 16#c9d3;
    GB2312[2100]:= 16#c4f3;
    GB2312[2101]:= 16#bee8;
    GB2312[2102]:= 16#b2b6;
    GB2312[2103]:= 16#c0cc;
    GB2312[2104]:= 16#cbf0;
    GB2312[2105]:= 16#bcf1;
    GB2312[2106]:= 16#bbbb;
    GB2312[2107]:= 16#b5b7;
    GB2312[2108]:= 16#c5f5;
    GB2312[2109]:= 16#dee6;
    GB2312[2110]:= 16#dee3;
    GB2312[2111]:= 16#bedd;
    GB2312[2112]:= 16#dedf;
    GB2312[2113]:= 16#b4b7;
    GB2312[2114]:= 16#bddd;
    GB2312[2115]:= 16#dee0;
    GB2312[2116]:= 16#c4ed;
    GB2312[2117]:= 16#cfc6;
    GB2312[2118]:= 16#b5e0;
    GB2312[2119]:= 16#b6de;
    GB2312[2120]:= 16#cada;
    GB2312[2121]:= 16#b5f4;
    GB2312[2122]:= 16#dee5;
    GB2312[2123]:= 16#d5c6;
    GB2312[2124]:= 16#dee1;
    GB2312[2125]:= 16#cccd;
    GB2312[2126]:= 16#c6fe;
    GB2312[2127]:= 16#c5c5;
    GB2312[2128]:= 16#d2b4;
    GB2312[2129]:= 16#bef2;
    GB2312[2130]:= 16#c2d3;
    GB2312[2131]:= 16#ccbd;
    GB2312[2132]:= 16#b3b8;
    GB2312[2133]:= 16#bdd3;
    GB2312[2134]:= 16#bfd8;
    GB2312[2135]:= 16#cdc6;
    GB2312[2136]:= 16#d1da;
    GB2312[2137]:= 16#b4eb;
    GB2312[2138]:= 16#dee4;
    GB2312[2139]:= 16#dedd;
    GB2312[2140]:= 16#dee7;
    GB2312[2141]:= 16#eafe;
    GB2312[2142]:= 16#c2b0;
    GB2312[2143]:= 16#dee2;
    GB2312[2144]:= 16#d6c0;
    GB2312[2145]:= 16#b5a7;
    GB2312[2146]:= 16#b2f4;
    GB2312[2147]:= 16#dee8;
    GB2312[2148]:= 16#def2;
    GB2312[2149]:= 16#deed;
    GB2312[2150]:= 16#def1;
    GB2312[2151]:= 16#c8e0;
    GB2312[2152]:= 16#d7e1;
    GB2312[2153]:= 16#deef;
    GB2312[2154]:= 16#c3e8;
    GB2312[2155]:= 16#cce1;
    GB2312[2156]:= 16#b2e5;
    GB2312[2157]:= 16#d2be;
    GB2312[2158]:= 16#deee;
    GB2312[2159]:= 16#deeb;
    GB2312[2160]:= 16#ced5;
    GB2312[2161]:= 16#b4a7;
    GB2312[2162]:= 16#bfab;
    GB2312[2163]:= 16#bebe;
    GB2312[2164]:= 16#bdd2;
    GB2312[2165]:= 16#dee9;
    GB2312[2166]:= 16#d4ae;
    GB2312[2167]:= 16#dede;
    GB2312[2168]:= 16#deea;
    GB2312[2169]:= 16#c0bf;
    GB2312[2170]:= 16#deec;
    GB2312[2171]:= 16#b2f3;
    GB2312[2172]:= 16#b8e9;
    GB2312[2173]:= 16#c2a7;
    GB2312[2174]:= 16#bdc1;
    GB2312[2175]:= 16#def5;
    GB2312[2176]:= 16#def8;
    GB2312[2177]:= 16#b2ab;
    GB2312[2178]:= 16#b4a4;
    GB2312[2179]:= 16#b4ea;
    GB2312[2180]:= 16#c9a6;
    GB2312[2181]:= 16#def6;
    GB2312[2182]:= 16#cbd1;
    GB2312[2183]:= 16#b8e3;
    GB2312[2184]:= 16#def7;
    GB2312[2185]:= 16#defa;
    GB2312[2186]:= 16#def9;
    GB2312[2187]:= 16#ccc2;
    GB2312[2188]:= 16#b0e1;
    GB2312[2189]:= 16#b4ee;
    GB2312[2190]:= 16#e5ba;
    GB2312[2191]:= 16#d0af;
    GB2312[2192]:= 16#b2eb;
    GB2312[2193]:= 16#eba1;
    GB2312[2194]:= 16#def4;
    GB2312[2195]:= 16#c9e3;
    GB2312[2196]:= 16#def3;
    GB2312[2197]:= 16#b0da;
    GB2312[2198]:= 16#d2a1;
    GB2312[2199]:= 16#b1f7;
    GB2312[2200]:= 16#ccaf;
    GB2312[2201]:= 16#def0;
    GB2312[2202]:= 16#cba4;
    GB2312[2203]:= 16#d5aa;
    GB2312[2204]:= 16#defb;
    GB2312[2205]:= 16#b4dd;
    GB2312[2206]:= 16#c4a6;
    GB2312[2207]:= 16#defd;
    GB2312[2208]:= 16#c3fe;
    GB2312[2209]:= 16#c4a1;
    GB2312[2210]:= 16#dfa1;
    GB2312[2211]:= 16#c1cc;
    GB2312[2212]:= 16#defc;
    GB2312[2213]:= 16#beef;
    GB2312[2214]:= 16#c6b2;
    GB2312[2215]:= 16#b3c5;
    GB2312[2216]:= 16#c8f6;
    GB2312[2217]:= 16#cbba;
    GB2312[2218]:= 16#defe;
    GB2312[2219]:= 16#dfa4;
    GB2312[2220]:= 16#d7b2;
    GB2312[2221]:= 16#b3b7;
    GB2312[2222]:= 16#c1c3;
    GB2312[2223]:= 16#c7cb;
    GB2312[2224]:= 16#b2a5;
    GB2312[2225]:= 16#b4e9;
    GB2312[2226]:= 16#d7ab;
    GB2312[2227]:= 16#c4ec;
    GB2312[2228]:= 16#dfa2;
    GB2312[2229]:= 16#dfa3;
    GB2312[2230]:= 16#dfa5;
    GB2312[2231]:= 16#bab3;
    GB2312[2232]:= 16#dfa6;
    GB2312[2233]:= 16#c0de;
    GB2312[2234]:= 16#c9c3;
    GB2312[2235]:= 16#b2d9;
    GB2312[2236]:= 16#c7e6;
    GB2312[2237]:= 16#dfa7;
    GB2312[2238]:= 16#c7dc;
    GB2312[2239]:= 16#dfa8;
    GB2312[2240]:= 16#eba2;
    GB2312[2241]:= 16#cbd3;
    GB2312[2242]:= 16#dfaa;
    GB2312[2243]:= 16#dfa9;
    GB2312[2244]:= 16#b2c1;
    GB2312[2245]:= 16#c5ca;
    GB2312[2246]:= 16#dfab;
    GB2312[2247]:= 16#d4dc;
    GB2312[2248]:= 16#c8c1;
    GB2312[2249]:= 16#dfac;
    GB2312[2250]:= 16#bef0;
    GB2312[2251]:= 16#dfad;
    GB2312[2252]:= 16#d6a7;
    GB2312[2253]:= 16#eab7;
    GB2312[2254]:= 16#ebb6;
    GB2312[2255]:= 16#cad5;
    GB2312[2256]:= 16#d8fc;
    GB2312[2257]:= 16#b8c4;
    GB2312[2258]:= 16#b9a5;
    GB2312[2259]:= 16#b7c5;
    GB2312[2260]:= 16#d5fe;
    GB2312[2261]:= 16#b9ca;
    GB2312[2262]:= 16#d0a7;
    GB2312[2263]:= 16#f4cd;
    GB2312[2264]:= 16#b5d0;
    GB2312[2265]:= 16#c3f4;
    GB2312[2266]:= 16#bec8;
    GB2312[2267]:= 16#ebb7;
    GB2312[2268]:= 16#b0bd;
    GB2312[2269]:= 16#bdcc;
    GB2312[2270]:= 16#c1b2;
    GB2312[2271]:= 16#b1d6;
    GB2312[2272]:= 16#b3a8;
    GB2312[2273]:= 16#b8d2;
    GB2312[2274]:= 16#c9a2;
    GB2312[2275]:= 16#b6d8;
    GB2312[2276]:= 16#ebb8;
    GB2312[2277]:= 16#beb4;
    GB2312[2278]:= 16#cafd;
    GB2312[2279]:= 16#c7c3;
    GB2312[2280]:= 16#d5fb;
    GB2312[2281]:= 16#b7f3;
    GB2312[2282]:= 16#cec4;
    GB2312[2283]:= 16#d5ab;
    GB2312[2284]:= 16#b1f3;
    GB2312[2285]:= 16#ecb3;
    GB2312[2286]:= 16#b0df;
    GB2312[2287]:= 16#ecb5;
    GB2312[2288]:= 16#b6b7;
    GB2312[2289]:= 16#c1cf;
    GB2312[2290]:= 16#f5fa;
    GB2312[2291]:= 16#d0b1;
    GB2312[2292]:= 16#d5e5;
    GB2312[2293]:= 16#ced3;
    GB2312[2294]:= 16#bdef;
    GB2312[2295]:= 16#b3e2;
    GB2312[2296]:= 16#b8ab;
    GB2312[2297]:= 16#d5b6;
    GB2312[2298]:= 16#edbd;
    GB2312[2299]:= 16#b6cf;
    GB2312[2300]:= 16#cbb9;
    GB2312[2301]:= 16#d0c2;
    GB2312[2302]:= 16#b7bd;
    GB2312[2303]:= 16#ecb6;
    GB2312[2304]:= 16#caa9;
    GB2312[2305]:= 16#c5d4;
    GB2312[2306]:= 16#ecb9;
    GB2312[2307]:= 16#ecb8;
    GB2312[2308]:= 16#c2c3;
    GB2312[2309]:= 16#ecb7;
    GB2312[2310]:= 16#d0fd;
    GB2312[2311]:= 16#ecba;
    GB2312[2312]:= 16#ecbb;
    GB2312[2313]:= 16#d7e5;
    GB2312[2314]:= 16#ecbc;
    GB2312[2315]:= 16#ecbd;
    GB2312[2316]:= 16#c6ec;
    GB2312[2317]:= 16#cede;
    GB2312[2318]:= 16#bcc8;
    GB2312[2319]:= 16#c8d5;
    GB2312[2320]:= 16#b5a9;
    GB2312[2321]:= 16#bec9;
    GB2312[2322]:= 16#d6bc;
    GB2312[2323]:= 16#d4e7;
    GB2312[2324]:= 16#d1ae;
    GB2312[2325]:= 16#d0f1;
    GB2312[2326]:= 16#eab8;
    GB2312[2327]:= 16#eab9;
    GB2312[2328]:= 16#eaba;
    GB2312[2329]:= 16#bab5;
    GB2312[2330]:= 16#cab1;
    GB2312[2331]:= 16#bff5;
    GB2312[2332]:= 16#cdfa;
    GB2312[2333]:= 16#eac0;
    GB2312[2334]:= 16#b0ba;
    GB2312[2335]:= 16#eabe;
    GB2312[2336]:= 16#c0a5;
    GB2312[2337]:= 16#eabb;
    GB2312[2338]:= 16#b2fd;
    GB2312[2339]:= 16#c3f7;
    GB2312[2340]:= 16#bbe8;
    GB2312[2341]:= 16#d2d7;
    GB2312[2342]:= 16#cef4;
    GB2312[2343]:= 16#eabf;
    GB2312[2344]:= 16#eabc;
    GB2312[2345]:= 16#eac3;
    GB2312[2346]:= 16#d0c7;
    GB2312[2347]:= 16#d3b3;
    GB2312[2348]:= 16#b4ba;
    GB2312[2349]:= 16#c3c1;
    GB2312[2350]:= 16#d7f2;
    GB2312[2351]:= 16#d5d1;
    GB2312[2352]:= 16#cac7;
    GB2312[2353]:= 16#eac5;
    GB2312[2354]:= 16#eac4;
    GB2312[2355]:= 16#eac7;
    GB2312[2356]:= 16#eac6;
    GB2312[2357]:= 16#d6e7;
    GB2312[2358]:= 16#cfd4;
    GB2312[2359]:= 16#eacb;
    GB2312[2360]:= 16#bbce;
    GB2312[2361]:= 16#bdfa;
    GB2312[2362]:= 16#c9ce;
    GB2312[2363]:= 16#eacc;
    GB2312[2364]:= 16#c9b9;
    GB2312[2365]:= 16#cffe;
    GB2312[2366]:= 16#eaca;
    GB2312[2367]:= 16#d4ce;
    GB2312[2368]:= 16#eacd;
    GB2312[2369]:= 16#eacf;
    GB2312[2370]:= 16#cded;
    GB2312[2371]:= 16#eac9;
    GB2312[2372]:= 16#eace;
    GB2312[2373]:= 16#ceee;
    GB2312[2374]:= 16#bbde;
    GB2312[2375]:= 16#b3bf;
    GB2312[2376]:= 16#c6d5;
    GB2312[2377]:= 16#beb0;
    GB2312[2378]:= 16#cefa;
    GB2312[2379]:= 16#c7e7;
    GB2312[2380]:= 16#bea7;
    GB2312[2381]:= 16#ead0;
    GB2312[2382]:= 16#d6c7;
    GB2312[2383]:= 16#c1c0;
    GB2312[2384]:= 16#d4dd;
    GB2312[2385]:= 16#ead1;
    GB2312[2386]:= 16#cfbe;
    GB2312[2387]:= 16#ead2;
    GB2312[2388]:= 16#caee;
    GB2312[2389]:= 16#c5af;
    GB2312[2390]:= 16#b0b5;
    GB2312[2391]:= 16#ead4;
    GB2312[2392]:= 16#ead3;
    GB2312[2393]:= 16#f4df;
    GB2312[2394]:= 16#c4ba;
    GB2312[2395]:= 16#b1a9;
    GB2312[2396]:= 16#e5df;
    GB2312[2397]:= 16#ead5;
    GB2312[2398]:= 16#caef;
    GB2312[2399]:= 16#ead6;
    GB2312[2400]:= 16#ead7;
    GB2312[2401]:= 16#c6d8;
    GB2312[2402]:= 16#ead8;
    GB2312[2403]:= 16#ead9;
    GB2312[2404]:= 16#d4bb;
    GB2312[2405]:= 16#c7fa;
    GB2312[2406]:= 16#d2b7;
    GB2312[2407]:= 16#b8fc;
    GB2312[2408]:= 16#eac2;
    GB2312[2409]:= 16#b2dc;
    GB2312[2410]:= 16#c2fc;
    GB2312[2411]:= 16#d4f8;
    GB2312[2412]:= 16#cce6;
    GB2312[2413]:= 16#d7ee;
    GB2312[2414]:= 16#d4c2;
    GB2312[2415]:= 16#d3d0;
    GB2312[2416]:= 16#ebc3;
    GB2312[2417]:= 16#c5f3;
    GB2312[2418]:= 16#b7fe;
    GB2312[2419]:= 16#ebd4;
    GB2312[2420]:= 16#cbb7;
    GB2312[2421]:= 16#ebde;
    GB2312[2422]:= 16#c0ca;
    GB2312[2423]:= 16#cdfb;
    GB2312[2424]:= 16#b3af;
    GB2312[2425]:= 16#c6da;
    GB2312[2426]:= 16#ebfc;
    GB2312[2427]:= 16#c4be;
    GB2312[2428]:= 16#ceb4;
    GB2312[2429]:= 16#c4a9;
    GB2312[2430]:= 16#b1be;
    GB2312[2431]:= 16#d4fd;
    GB2312[2432]:= 16#caf5;
    GB2312[2433]:= 16#d6ec;
    GB2312[2434]:= 16#c6d3;
    GB2312[2435]:= 16#b6e4;
    GB2312[2436]:= 16#bbfa;
    GB2312[2437]:= 16#d0e0;
    GB2312[2438]:= 16#c9b1;
    GB2312[2439]:= 16#d4d3;
    GB2312[2440]:= 16#c8a8;
    GB2312[2441]:= 16#b8cb;
    GB2312[2442]:= 16#e8be;
    GB2312[2443]:= 16#c9bc;
    GB2312[2444]:= 16#e8bb;
    GB2312[2445]:= 16#c0ee;
    GB2312[2446]:= 16#d0d3;
    GB2312[2447]:= 16#b2c4;
    GB2312[2448]:= 16#b4e5;
    GB2312[2449]:= 16#e8bc;
    GB2312[2450]:= 16#d5c8;
    GB2312[2451]:= 16#b6c5;
    GB2312[2452]:= 16#e8bd;
    GB2312[2453]:= 16#caf8;
    GB2312[2454]:= 16#b8dc;
    GB2312[2455]:= 16#ccf5;
    GB2312[2456]:= 16#c0b4;
    GB2312[2457]:= 16#d1ee;
    GB2312[2458]:= 16#e8bf;
    GB2312[2459]:= 16#e8c2;
    GB2312[2460]:= 16#babc;
    GB2312[2461]:= 16#b1ad;
    GB2312[2462]:= 16#bddc;
    GB2312[2463]:= 16#eabd;
    GB2312[2464]:= 16#e8c3;
    GB2312[2465]:= 16#e8c6;
    GB2312[2466]:= 16#e8cb;
    GB2312[2467]:= 16#e8cc;
    GB2312[2468]:= 16#cbc9;
    GB2312[2469]:= 16#b0e5;
    GB2312[2470]:= 16#bcab;
    GB2312[2471]:= 16#b9b9;
    GB2312[2472]:= 16#e8c1;
    GB2312[2473]:= 16#cdf7;
    GB2312[2474]:= 16#e8ca;
    GB2312[2475]:= 16#cef6;
    GB2312[2476]:= 16#d5ed;
    GB2312[2477]:= 16#c1d6;
    GB2312[2478]:= 16#e8c4;
    GB2312[2479]:= 16#c3b6;
    GB2312[2480]:= 16#b9fb;
    GB2312[2481]:= 16#d6a6;
    GB2312[2482]:= 16#e8c8;
    GB2312[2483]:= 16#cae0;
    GB2312[2484]:= 16#d4e6;
    GB2312[2485]:= 16#e8c0;
    GB2312[2486]:= 16#e8c5;
    GB2312[2487]:= 16#e8c7;
    GB2312[2488]:= 16#c7b9;
    GB2312[2489]:= 16#b7e3;
    GB2312[2490]:= 16#e8c9;
    GB2312[2491]:= 16#bfdd;
    GB2312[2492]:= 16#e8d2;
    GB2312[2493]:= 16#e8d7;
    GB2312[2494]:= 16#e8d5;
    GB2312[2495]:= 16#bcdc;
    GB2312[2496]:= 16#bccf;
    GB2312[2497]:= 16#e8db;
    GB2312[2498]:= 16#e8de;
    GB2312[2499]:= 16#e8da;
    GB2312[2500]:= 16#b1fa;
    GB2312[2501]:= 16#b0d8;
    GB2312[2502]:= 16#c4b3;
    GB2312[2503]:= 16#b8cc;
    GB2312[2504]:= 16#c6e2;
    GB2312[2505]:= 16#c8be;
    GB2312[2506]:= 16#c8e1;
    GB2312[2507]:= 16#e8cf;
    GB2312[2508]:= 16#e8d4;
    GB2312[2509]:= 16#e8d6;
    GB2312[2510]:= 16#b9f1;
    GB2312[2511]:= 16#e8d8;
    GB2312[2512]:= 16#d7f5;
    GB2312[2513]:= 16#c4fb;
    GB2312[2514]:= 16#e8dc;
    GB2312[2515]:= 16#b2e9;
    GB2312[2516]:= 16#e8d1;
    GB2312[2517]:= 16#bced;
    GB2312[2518]:= 16#bfc2;
    GB2312[2519]:= 16#e8cd;
    GB2312[2520]:= 16#d6f9;
    GB2312[2521]:= 16#c1f8;
    GB2312[2522]:= 16#b2f1;
    GB2312[2523]:= 16#e8df;
    GB2312[2524]:= 16#cac1;
    GB2312[2525]:= 16#e8d9;
    GB2312[2526]:= 16#d5a4;
    GB2312[2527]:= 16#b1ea;
    GB2312[2528]:= 16#d5bb;
    GB2312[2529]:= 16#e8ce;
    GB2312[2530]:= 16#e8d0;
    GB2312[2531]:= 16#b6b0;
    GB2312[2532]:= 16#e8d3;
    GB2312[2533]:= 16#e8dd;
    GB2312[2534]:= 16#c0b8;
    GB2312[2535]:= 16#caf7;
    GB2312[2536]:= 16#cba8;
    GB2312[2537]:= 16#c6dc;
    GB2312[2538]:= 16#c0f5;
    GB2312[2539]:= 16#e8e9;
    GB2312[2540]:= 16#d0a3;
    GB2312[2541]:= 16#e8f2;
    GB2312[2542]:= 16#d6ea;
    GB2312[2543]:= 16#e8e0;
    GB2312[2544]:= 16#e8e1;
    GB2312[2545]:= 16#d1f9;
    GB2312[2546]:= 16#bacb;
    GB2312[2547]:= 16#b8f9;
    GB2312[2548]:= 16#b8f1;
    GB2312[2549]:= 16#d4d4;
    GB2312[2550]:= 16#e8ef;
    GB2312[2551]:= 16#e8ee;
    GB2312[2552]:= 16#e8ec;
    GB2312[2553]:= 16#b9f0;
    GB2312[2554]:= 16#ccd2;
    GB2312[2555]:= 16#e8e6;
    GB2312[2556]:= 16#cea6;
    GB2312[2557]:= 16#bff2;
    GB2312[2558]:= 16#b0b8;
    GB2312[2559]:= 16#e8f1;
    GB2312[2560]:= 16#e8f0;
    GB2312[2561]:= 16#d7c0;
    GB2312[2562]:= 16#e8e4;
    GB2312[2563]:= 16#cda9;
    GB2312[2564]:= 16#c9a3;
    GB2312[2565]:= 16#bbb8;
    GB2312[2566]:= 16#bddb;
    GB2312[2567]:= 16#e8ea;
    GB2312[2568]:= 16#e8e2;
    GB2312[2569]:= 16#e8e3;
    GB2312[2570]:= 16#e8e5;
    GB2312[2571]:= 16#b5b5;
    GB2312[2572]:= 16#e8e7;
    GB2312[2573]:= 16#c7c5;
    GB2312[2574]:= 16#e8eb;
    GB2312[2575]:= 16#e8ed;
    GB2312[2576]:= 16#bdb0;
    GB2312[2577]:= 16#d7ae;
    GB2312[2578]:= 16#e8f8;
    GB2312[2579]:= 16#e8f5;
    GB2312[2580]:= 16#cdb0;
    GB2312[2581]:= 16#e8f6;
    GB2312[2582]:= 16#c1ba;
    GB2312[2583]:= 16#e8e8;
    GB2312[2584]:= 16#c3b7;
    GB2312[2585]:= 16#b0f0;
    GB2312[2586]:= 16#e8f4;
    GB2312[2587]:= 16#e8f7;
    GB2312[2588]:= 16#b9a3;
    GB2312[2589]:= 16#c9d2;
    GB2312[2590]:= 16#c3ce;
    GB2312[2591]:= 16#cee0;
    GB2312[2592]:= 16#c0e6;
    GB2312[2593]:= 16#cbf3;
    GB2312[2594]:= 16#ccdd;
    GB2312[2595]:= 16#d0b5;
    GB2312[2596]:= 16#cae1;
    GB2312[2597]:= 16#e8f3;
    GB2312[2598]:= 16#bcec;
    GB2312[2599]:= 16#e8f9;
    GB2312[2600]:= 16#c3de;
    GB2312[2601]:= 16#c6e5;
    GB2312[2602]:= 16#b9f7;
    GB2312[2603]:= 16#b0f4;
    GB2312[2604]:= 16#d7d8;
    GB2312[2605]:= 16#bcac;
    GB2312[2606]:= 16#c5ef;
    GB2312[2607]:= 16#ccc4;
    GB2312[2608]:= 16#e9a6;
    GB2312[2609]:= 16#c9ad;
    GB2312[2610]:= 16#e9a2;
    GB2312[2611]:= 16#c0e2;
    GB2312[2612]:= 16#bfc3;
    GB2312[2613]:= 16#e8fe;
    GB2312[2614]:= 16#b9d7;
    GB2312[2615]:= 16#e8fb;
    GB2312[2616]:= 16#e9a4;
    GB2312[2617]:= 16#d2ce;
    GB2312[2618]:= 16#e9a3;
    GB2312[2619]:= 16#d6b2;
    GB2312[2620]:= 16#d7b5;
    GB2312[2621]:= 16#e9a7;
    GB2312[2622]:= 16#bdb7;
    GB2312[2623]:= 16#e8fc;
    GB2312[2624]:= 16#e8fd;
    GB2312[2625]:= 16#e9a1;
    GB2312[2626]:= 16#cdd6;
    GB2312[2627]:= 16#d2ac;
    GB2312[2628]:= 16#e9b2;
    GB2312[2629]:= 16#e9a9;
    GB2312[2630]:= 16#b4aa;
    GB2312[2631]:= 16#b4bb;
    GB2312[2632]:= 16#e9ab;
    GB2312[2633]:= 16#d0a8;
    GB2312[2634]:= 16#e9a5;
    GB2312[2635]:= 16#b3fe;
    GB2312[2636]:= 16#e9ac;
    GB2312[2637]:= 16#c0e3;
    GB2312[2638]:= 16#e9aa;
    GB2312[2639]:= 16#e9b9;
    GB2312[2640]:= 16#e9b8;
    GB2312[2641]:= 16#e9ae;
    GB2312[2642]:= 16#e8fa;
    GB2312[2643]:= 16#e9a8;
    GB2312[2644]:= 16#bfac;
    GB2312[2645]:= 16#e9b1;
    GB2312[2646]:= 16#e9ba;
    GB2312[2647]:= 16#c2a5;
    GB2312[2648]:= 16#e9af;
    GB2312[2649]:= 16#b8c5;
    GB2312[2650]:= 16#e9ad;
    GB2312[2651]:= 16#d3dc;
    GB2312[2652]:= 16#e9b4;
    GB2312[2653]:= 16#e9b5;
    GB2312[2654]:= 16#e9b7;
    GB2312[2655]:= 16#e9c7;
    GB2312[2656]:= 16#c0c6;
    GB2312[2657]:= 16#e9c5;
    GB2312[2658]:= 16#e9b0;
    GB2312[2659]:= 16#e9bb;
    GB2312[2660]:= 16#b0f1;
    GB2312[2661]:= 16#e9bc;
    GB2312[2662]:= 16#d5a5;
    GB2312[2663]:= 16#e9be;
    GB2312[2664]:= 16#e9bf;
    GB2312[2665]:= 16#e9c1;
    GB2312[2666]:= 16#c1f1;
    GB2312[2667]:= 16#c8b6;
    GB2312[2668]:= 16#e9bd;
    GB2312[2669]:= 16#e9c2;
    GB2312[2670]:= 16#e9c3;
    GB2312[2671]:= 16#e9b3;
    GB2312[2672]:= 16#e9b6;
    GB2312[2673]:= 16#bbb1;
    GB2312[2674]:= 16#e9c0;
    GB2312[2675]:= 16#bcf7;
    GB2312[2676]:= 16#e9c4;
    GB2312[2677]:= 16#e9c6;
    GB2312[2678]:= 16#e9ca;
    GB2312[2679]:= 16#e9ce;
    GB2312[2680]:= 16#b2db;
    GB2312[2681]:= 16#e9c8;
    GB2312[2682]:= 16#b7ae;
    GB2312[2683]:= 16#e9cb;
    GB2312[2684]:= 16#e9cc;
    GB2312[2685]:= 16#d5c1;
    GB2312[2686]:= 16#c4a3;
    GB2312[2687]:= 16#e9d8;
    GB2312[2688]:= 16#bae1;
    GB2312[2689]:= 16#e9c9;
    GB2312[2690]:= 16#d3a3;
    GB2312[2691]:= 16#e9d4;
    GB2312[2692]:= 16#e9d7;
    GB2312[2693]:= 16#e9d0;
    GB2312[2694]:= 16#e9cf;
    GB2312[2695]:= 16#c7c1;
    GB2312[2696]:= 16#e9d2;
    GB2312[2697]:= 16#e9d9;
    GB2312[2698]:= 16#b3c8;
    GB2312[2699]:= 16#e9d3;
    GB2312[2700]:= 16#cff0;
    GB2312[2701]:= 16#e9cd;
    GB2312[2702]:= 16#b3f7;
    GB2312[2703]:= 16#e9d6;
    GB2312[2704]:= 16#e9da;
    GB2312[2705]:= 16#ccb4;
    GB2312[2706]:= 16#cfad;
    GB2312[2707]:= 16#e9d5;
    GB2312[2708]:= 16#e9dc;
    GB2312[2709]:= 16#e9db;
    GB2312[2710]:= 16#e9de;
    GB2312[2711]:= 16#e9d1;
    GB2312[2712]:= 16#e9dd;
    GB2312[2713]:= 16#e9df;
    GB2312[2714]:= 16#c3ca;
    GB2312[2715]:= 16#c7b7;
    GB2312[2716]:= 16#b4ce;
    GB2312[2717]:= 16#bbb6;
    GB2312[2718]:= 16#d0c0;
    GB2312[2719]:= 16#eca3;
    GB2312[2720]:= 16#c5b7;
    GB2312[2721]:= 16#d3fb;
    GB2312[2722]:= 16#eca4;
    GB2312[2723]:= 16#eca5;
    GB2312[2724]:= 16#c6db;
    GB2312[2725]:= 16#bfee;
    GB2312[2726]:= 16#eca6;
    GB2312[2727]:= 16#eca7;
    GB2312[2728]:= 16#d0aa;
    GB2312[2729]:= 16#c7b8;
    GB2312[2730]:= 16#b8e8;
    GB2312[2731]:= 16#eca8;
    GB2312[2732]:= 16#d6b9;
    GB2312[2733]:= 16#d5fd;
    GB2312[2734]:= 16#b4cb;
    GB2312[2735]:= 16#b2bd;
    GB2312[2736]:= 16#cee4;
    GB2312[2737]:= 16#c6e7;
    GB2312[2738]:= 16#cde1;
    GB2312[2739]:= 16#b4f5;
    GB2312[2740]:= 16#cbc0;
    GB2312[2741]:= 16#bcdf;
    GB2312[2742]:= 16#e9e2;
    GB2312[2743]:= 16#e9e3;
    GB2312[2744]:= 16#d1ea;
    GB2312[2745]:= 16#e9e5;
    GB2312[2746]:= 16#b4f9;
    GB2312[2747]:= 16#e9e4;
    GB2312[2748]:= 16#d1b3;
    GB2312[2749]:= 16#cae2;
    GB2312[2750]:= 16#b2d0;
    GB2312[2751]:= 16#e9e8;
    GB2312[2752]:= 16#e9e6;
    GB2312[2753]:= 16#e9e7;
    GB2312[2754]:= 16#d6b3;
    GB2312[2755]:= 16#e9e9;
    GB2312[2756]:= 16#e9ea;
    GB2312[2757]:= 16#e9eb;
    GB2312[2758]:= 16#e9ec;
    GB2312[2759]:= 16#ecaf;
    GB2312[2760]:= 16#c5b9;
    GB2312[2761]:= 16#b6ce;
    GB2312[2762]:= 16#d2f3;
    GB2312[2763]:= 16#b5ee;
    GB2312[2764]:= 16#bbd9;
    GB2312[2765]:= 16#ecb1;
    GB2312[2766]:= 16#d2e3;
    GB2312[2767]:= 16#cee3;
    GB2312[2768]:= 16#c4b8;
    GB2312[2769]:= 16#c3bf;
    GB2312[2770]:= 16#b6be;
    GB2312[2771]:= 16#d8b9;
    GB2312[2772]:= 16#b1c8;
    GB2312[2773]:= 16#b1cf;
    GB2312[2774]:= 16#b1d1;
    GB2312[2775]:= 16#c5fe;
    GB2312[2776]:= 16#b1d0;
    GB2312[2777]:= 16#c3ab;
    GB2312[2778]:= 16#d5b1;
    GB2312[2779]:= 16#eba4;
    GB2312[2780]:= 16#bac1;
    GB2312[2781]:= 16#ccba;
    GB2312[2782]:= 16#eba5;
    GB2312[2783]:= 16#eba7;
    GB2312[2784]:= 16#eba8;
    GB2312[2785]:= 16#eba6;
    GB2312[2786]:= 16#eba9;
    GB2312[2787]:= 16#ebab;
    GB2312[2788]:= 16#ebaa;
    GB2312[2789]:= 16#ebac;
    GB2312[2790]:= 16#cacf;
    GB2312[2791]:= 16#d8b5;
    GB2312[2792]:= 16#c3f1;
    GB2312[2793]:= 16#c3a5;
    GB2312[2794]:= 16#c6f8;
    GB2312[2795]:= 16#ebad;
    GB2312[2796]:= 16#c4ca;
    GB2312[2797]:= 16#ebae;
    GB2312[2798]:= 16#ebaf;
    GB2312[2799]:= 16#ebb0;
    GB2312[2800]:= 16#b7d5;
    GB2312[2801]:= 16#b7fa;
    GB2312[2802]:= 16#ebb1;
    GB2312[2803]:= 16#c7e2;
    GB2312[2804]:= 16#ebb3;
    GB2312[2805]:= 16#baa4;
    GB2312[2806]:= 16#d1f5;
    GB2312[2807]:= 16#b0b1;
    GB2312[2808]:= 16#ebb2;
    GB2312[2809]:= 16#ebb4;
    GB2312[2810]:= 16#b5aa;
    GB2312[2811]:= 16#c2c8;
    GB2312[2812]:= 16#c7e8;
    GB2312[2813]:= 16#ebb5;
    GB2312[2814]:= 16#cbae;
    GB2312[2815]:= 16#e3df;
    GB2312[2816]:= 16#d3c0;
    GB2312[2817]:= 16#d9db;
    GB2312[2818]:= 16#cda1;
    GB2312[2819]:= 16#d6ad;
    GB2312[2820]:= 16#c7f3;
    GB2312[2821]:= 16#d9e0;
    GB2312[2822]:= 16#bbe3;
    GB2312[2823]:= 16#baba;
    GB2312[2824]:= 16#e3e2;
    GB2312[2825]:= 16#cfab;
    GB2312[2826]:= 16#e3e0;
    GB2312[2827]:= 16#c9c7;
    GB2312[2828]:= 16#bab9;
    GB2312[2829]:= 16#d1b4;
    GB2312[2830]:= 16#e3e1;
    GB2312[2831]:= 16#c8ea;
    GB2312[2832]:= 16#b9af;
    GB2312[2833]:= 16#bdad;
    GB2312[2834]:= 16#b3d8;
    GB2312[2835]:= 16#cedb;
    GB2312[2836]:= 16#ccc0;
    GB2312[2837]:= 16#e3e8;
    GB2312[2838]:= 16#e3e9;
    GB2312[2839]:= 16#cdf4;
    GB2312[2840]:= 16#ccad;
    GB2312[2841]:= 16#bcb3;
    GB2312[2842]:= 16#e3ea;
    GB2312[2843]:= 16#e3eb;
    GB2312[2844]:= 16#d0da;
    GB2312[2845]:= 16#c6fb;
    GB2312[2846]:= 16#b7da;
    GB2312[2847]:= 16#c7df;
    GB2312[2848]:= 16#d2ca;
    GB2312[2849]:= 16#ced6;
    GB2312[2850]:= 16#e3e4;
    GB2312[2851]:= 16#e3ec;
    GB2312[2852]:= 16#c9f2;
    GB2312[2853]:= 16#b3c1;
    GB2312[2854]:= 16#e3e7;
    GB2312[2855]:= 16#c6e3;
    GB2312[2856]:= 16#e3e5;
    GB2312[2857]:= 16#edb3;
    GB2312[2858]:= 16#e3e6;
    GB2312[2859]:= 16#c9b3;
    GB2312[2860]:= 16#c5e6;
    GB2312[2861]:= 16#b9b5;
    GB2312[2862]:= 16#c3bb;
    GB2312[2863]:= 16#e3e3;
    GB2312[2864]:= 16#c5bd;
    GB2312[2865]:= 16#c1a4;
    GB2312[2866]:= 16#c2d9;
    GB2312[2867]:= 16#b2d7;
    GB2312[2868]:= 16#e3ed;
    GB2312[2869]:= 16#bba6;
    GB2312[2870]:= 16#c4ad;
    GB2312[2871]:= 16#e3f0;
    GB2312[2872]:= 16#beda;
    GB2312[2873]:= 16#e3fb;
    GB2312[2874]:= 16#e3f5;
    GB2312[2875]:= 16#bad3;
    GB2312[2876]:= 16#b7d0;
    GB2312[2877]:= 16#d3cd;
    GB2312[2878]:= 16#d6ce;
    GB2312[2879]:= 16#d5d3;
    GB2312[2880]:= 16#b9c1;
    GB2312[2881]:= 16#d5b4;
    GB2312[2882]:= 16#d1d8;
    GB2312[2883]:= 16#d0b9;
    GB2312[2884]:= 16#c7f6;
    GB2312[2885]:= 16#c8aa;
    GB2312[2886]:= 16#b2b4;
    GB2312[2887]:= 16#c3da;
    GB2312[2888]:= 16#e3ee;
    GB2312[2889]:= 16#e3fc;
    GB2312[2890]:= 16#e3ef;
    GB2312[2891]:= 16#b7a8;
    GB2312[2892]:= 16#e3f7;
    GB2312[2893]:= 16#e3f4;
    GB2312[2894]:= 16#b7ba;
    GB2312[2895]:= 16#c5a2;
    GB2312[2896]:= 16#e3f6;
    GB2312[2897]:= 16#c5dd;
    GB2312[2898]:= 16#b2a8;
    GB2312[2899]:= 16#c6fc;
    GB2312[2900]:= 16#c4e0;
    GB2312[2901]:= 16#d7a2;
    GB2312[2902]:= 16#c0e1;
    GB2312[2903]:= 16#e3f9;
    GB2312[2904]:= 16#e3fa;
    GB2312[2905]:= 16#e3fd;
    GB2312[2906]:= 16#cca9;
    GB2312[2907]:= 16#e3f3;
    GB2312[2908]:= 16#d3be;
    GB2312[2909]:= 16#b1c3;
    GB2312[2910]:= 16#edb4;
    GB2312[2911]:= 16#e3f1;
    GB2312[2912]:= 16#e3f2;
    GB2312[2913]:= 16#e3f8;
    GB2312[2914]:= 16#d0ba;
    GB2312[2915]:= 16#c6c3;
    GB2312[2916]:= 16#d4f3;
    GB2312[2917]:= 16#e3fe;
    GB2312[2918]:= 16#bde0;
    GB2312[2919]:= 16#e4a7;
    GB2312[2920]:= 16#e4a6;
    GB2312[2921]:= 16#d1f3;
    GB2312[2922]:= 16#e4a3;
    GB2312[2923]:= 16#e4a9;
    GB2312[2924]:= 16#c8f7;
    GB2312[2925]:= 16#cfb4;
    GB2312[2926]:= 16#e4a8;
    GB2312[2927]:= 16#e4ae;
    GB2312[2928]:= 16#c2e5;
    GB2312[2929]:= 16#b6b4;
    GB2312[2930]:= 16#bdf2;
    GB2312[2931]:= 16#e4a2;
    GB2312[2932]:= 16#bae9;
    GB2312[2933]:= 16#e4aa;
    GB2312[2934]:= 16#e4ac;
    GB2312[2935]:= 16#b6fd;
    GB2312[2936]:= 16#d6de;
    GB2312[2937]:= 16#e4b2;
    GB2312[2938]:= 16#e4ad;
    GB2312[2939]:= 16#e4a1;
    GB2312[2940]:= 16#bbee;
    GB2312[2941]:= 16#cddd;
    GB2312[2942]:= 16#c7a2;
    GB2312[2943]:= 16#c5c9;
    GB2312[2944]:= 16#c1f7;
    GB2312[2945]:= 16#e4a4;
    GB2312[2946]:= 16#c7b3;
    GB2312[2947]:= 16#bdac;
    GB2312[2948]:= 16#bdbd;
    GB2312[2949]:= 16#e4a5;
    GB2312[2950]:= 16#d7c7;
    GB2312[2951]:= 16#b2e2;
    GB2312[2952]:= 16#e4ab;
    GB2312[2953]:= 16#bcc3;
    GB2312[2954]:= 16#e4af;
    GB2312[2955]:= 16#bbeb;
    GB2312[2956]:= 16#e4b0;
    GB2312[2957]:= 16#c5a8;
    GB2312[2958]:= 16#e4b1;
    GB2312[2959]:= 16#d5e3;
    GB2312[2960]:= 16#bfa3;
    GB2312[2961]:= 16#e4ba;
    GB2312[2962]:= 16#e4b7;
    GB2312[2963]:= 16#e4bb;
    GB2312[2964]:= 16#e4bd;
    GB2312[2965]:= 16#c6d6;
    GB2312[2966]:= 16#bac6;
    GB2312[2967]:= 16#c0cb;
    GB2312[2968]:= 16#b8a1;
    GB2312[2969]:= 16#e4b4;
    GB2312[2970]:= 16#d4a1;
    GB2312[2971]:= 16#baa3;
    GB2312[2972]:= 16#bdfe;
    GB2312[2973]:= 16#e4bc;
    GB2312[2974]:= 16#cdbf;
    GB2312[2975]:= 16#c4f9;
    GB2312[2976]:= 16#cffb;
    GB2312[2977]:= 16#c9e6;
    GB2312[2978]:= 16#d3bf;
    GB2312[2979]:= 16#cfd1;
    GB2312[2980]:= 16#e4b3;
    GB2312[2981]:= 16#e4b8;
    GB2312[2982]:= 16#e4b9;
    GB2312[2983]:= 16#cce9;
    GB2312[2984]:= 16#ccce;
    GB2312[2985]:= 16#c0d4;
    GB2312[2986]:= 16#e4b5;
    GB2312[2987]:= 16#c1b0;
    GB2312[2988]:= 16#e4b6;
    GB2312[2989]:= 16#ced0;
    GB2312[2990]:= 16#bbc1;
    GB2312[2991]:= 16#b5d3;
    GB2312[2992]:= 16#c8f3;
    GB2312[2993]:= 16#bda7;
    GB2312[2994]:= 16#d5c7;
    GB2312[2995]:= 16#c9ac;
    GB2312[2996]:= 16#b8a2;
    GB2312[2997]:= 16#e4ca;
    GB2312[2998]:= 16#e4cc;
    GB2312[2999]:= 16#d1c4;     //GB2312码 2000-2999
END_IF;
(* Rung 14 *)
IF P_On THEN
    GB2312[3000]:= 16#d2ba;
    GB2312[3001]:= 16#baad;
    GB2312[3002]:= 16#bad4;
    GB2312[3003]:= 16#e4c3;
    GB2312[3004]:= 16#b5ed;
    GB2312[3005]:= 16#d7cd;
    GB2312[3006]:= 16#e4c0;
    GB2312[3007]:= 16#cffd;
    GB2312[3008]:= 16#e4bf;
    GB2312[3009]:= 16#c1dc;
    GB2312[3010]:= 16#ccca;
    GB2312[3011]:= 16#cae7;
    GB2312[3012]:= 16#c4d7;
    GB2312[3013]:= 16#ccd4;
    GB2312[3014]:= 16#e4c8;
    GB2312[3015]:= 16#e4c7;
    GB2312[3016]:= 16#e4c1;
    GB2312[3017]:= 16#e4c4;
    GB2312[3018]:= 16#b5ad;
    GB2312[3019]:= 16#d3d9;
    GB2312[3020]:= 16#e4c6;
    GB2312[3021]:= 16#d2f9;
    GB2312[3022]:= 16#b4e3;
    GB2312[3023]:= 16#bbb4;
    GB2312[3024]:= 16#c9ee;
    GB2312[3025]:= 16#b4be;
    GB2312[3026]:= 16#bbec;
    GB2312[3027]:= 16#d1cd;
    GB2312[3028]:= 16#cced;
    GB2312[3029]:= 16#edb5;
    GB2312[3030]:= 16#c7e5;
    GB2312[3031]:= 16#d4a8;
    GB2312[3032]:= 16#e4cb;
    GB2312[3033]:= 16#d7d5;
    GB2312[3034]:= 16#e4c2;
    GB2312[3035]:= 16#bda5;
    GB2312[3036]:= 16#e4c5;
    GB2312[3037]:= 16#d3e6;
    GB2312[3038]:= 16#e4c9;
    GB2312[3039]:= 16#c9f8;
    GB2312[3040]:= 16#e4be;
    GB2312[3041]:= 16#d3e5;
    GB2312[3042]:= 16#c7fe;
    GB2312[3043]:= 16#b6c9;
    GB2312[3044]:= 16#d4fc;
    GB2312[3045]:= 16#b2b3;
    GB2312[3046]:= 16#e4d7;
    GB2312[3047]:= 16#cec2;
    GB2312[3048]:= 16#e4cd;
    GB2312[3049]:= 16#cebc;
    GB2312[3050]:= 16#b8db;
    GB2312[3051]:= 16#e4d6;
    GB2312[3052]:= 16#bfca;
    GB2312[3053]:= 16#d3ce;
    GB2312[3054]:= 16#c3ec;
    GB2312[3055]:= 16#c5c8;
    GB2312[3056]:= 16#e4d8;
    GB2312[3057]:= 16#cdc4;
    GB2312[3058]:= 16#e4cf;
    GB2312[3059]:= 16#e4d4;
    GB2312[3060]:= 16#e4d5;
    GB2312[3061]:= 16#bafe;
    GB2312[3062]:= 16#cfe6;
    GB2312[3063]:= 16#d5bf;
    GB2312[3064]:= 16#e4d2;
    GB2312[3065]:= 16#e4d0;
    GB2312[3066]:= 16#e4ce;
    GB2312[3067]:= 16#cde5;
    GB2312[3068]:= 16#caaa;
    GB2312[3069]:= 16#c0a3;
    GB2312[3070]:= 16#bda6;
    GB2312[3071]:= 16#e4d3;
    GB2312[3072]:= 16#b8c8;
    GB2312[3073]:= 16#e4e7;
    GB2312[3074]:= 16#d4b4;
    GB2312[3075]:= 16#e4db;
    GB2312[3076]:= 16#c1ef;
    GB2312[3077]:= 16#e4e9;
    GB2312[3078]:= 16#d2e7;
    GB2312[3079]:= 16#e4df;
    GB2312[3080]:= 16#e4e0;
    GB2312[3081]:= 16#cfaa;
    GB2312[3082]:= 16#cbdd;
    GB2312[3083]:= 16#e4da;
    GB2312[3084]:= 16#e4d1;
    GB2312[3085]:= 16#e4e5;
    GB2312[3086]:= 16#c8dc;
    GB2312[3087]:= 16#e4e3;
    GB2312[3088]:= 16#c4e7;
    GB2312[3089]:= 16#e4e2;
    GB2312[3090]:= 16#e4e1;
    GB2312[3091]:= 16#b3fc;
    GB2312[3092]:= 16#e4e8;
    GB2312[3093]:= 16#b5e1;
    GB2312[3094]:= 16#d7cc;
    GB2312[3095]:= 16#e4e6;
    GB2312[3096]:= 16#bbac;
    GB2312[3097]:= 16#d7d2;
    GB2312[3098]:= 16#cccf;
    GB2312[3099]:= 16#ebf8;
    GB2312[3100]:= 16#e4e4;
    GB2312[3101]:= 16#b9f6;
    GB2312[3102]:= 16#d6cd;
    GB2312[3103]:= 16#e4d9;
    GB2312[3104]:= 16#e4dc;
    GB2312[3105]:= 16#c2fa;
    GB2312[3106]:= 16#e4de;
    GB2312[3107]:= 16#c2cb;
    GB2312[3108]:= 16#c0c4;
    GB2312[3109]:= 16#c2d0;
    GB2312[3110]:= 16#b1f5;
    GB2312[3111]:= 16#ccb2;
    GB2312[3112]:= 16#b5ce;
    GB2312[3113]:= 16#e4ef;
    GB2312[3114]:= 16#c6af;
    GB2312[3115]:= 16#c6e1;
    GB2312[3116]:= 16#e4f5;
    GB2312[3117]:= 16#c2a9;
    GB2312[3118]:= 16#c0ec;
    GB2312[3119]:= 16#d1dd;
    GB2312[3120]:= 16#e4ee;
    GB2312[3121]:= 16#c4ae;
    GB2312[3122]:= 16#e4ed;
    GB2312[3123]:= 16#e4f6;
    GB2312[3124]:= 16#e4f4;
    GB2312[3125]:= 16#c2fe;
    GB2312[3126]:= 16#e4dd;
    GB2312[3127]:= 16#e4f0;
    GB2312[3128]:= 16#cafe;
    GB2312[3129]:= 16#d5c4;
    GB2312[3130]:= 16#e4f1;
    GB2312[3131]:= 16#d1fa;
    GB2312[3132]:= 16#e4eb;
    GB2312[3133]:= 16#e4ec;
    GB2312[3134]:= 16#e4f2;
    GB2312[3135]:= 16#ceab;
    GB2312[3136]:= 16#c5cb;
    GB2312[3137]:= 16#c7b1;
    GB2312[3138]:= 16#c2ba;
    GB2312[3139]:= 16#e4ea;
    GB2312[3140]:= 16#c1ca;
    GB2312[3141]:= 16#ccb6;
    GB2312[3142]:= 16#b3b1;
    GB2312[3143]:= 16#e4fb;
    GB2312[3144]:= 16#e4f3;
    GB2312[3145]:= 16#e4fa;
    GB2312[3146]:= 16#e4fd;
    GB2312[3147]:= 16#e4fc;
    GB2312[3148]:= 16#b3ce;
    GB2312[3149]:= 16#b3ba;
    GB2312[3150]:= 16#e4f7;
    GB2312[3151]:= 16#e4f9;
    GB2312[3152]:= 16#e4f8;
    GB2312[3153]:= 16#c5ec;
    GB2312[3154]:= 16#c0bd;
    GB2312[3155]:= 16#d4e8;
    GB2312[3156]:= 16#e5a2;
    GB2312[3157]:= 16#b0c4;
    GB2312[3158]:= 16#e5a4;
    GB2312[3159]:= 16#e5a3;
    GB2312[3160]:= 16#bca4;
    GB2312[3161]:= 16#e5a5;
    GB2312[3162]:= 16#e5a1;
    GB2312[3163]:= 16#e4fe;
    GB2312[3164]:= 16#b1f4;
    GB2312[3165]:= 16#e5a8;
    GB2312[3166]:= 16#e5a9;
    GB2312[3167]:= 16#e5a6;
    GB2312[3168]:= 16#e5a7;
    GB2312[3169]:= 16#e5aa;
    GB2312[3170]:= 16#c6d9;
    GB2312[3171]:= 16#e5ab;
    GB2312[3172]:= 16#e5ad;
    GB2312[3173]:= 16#e5ac;
    GB2312[3174]:= 16#e5af;
    GB2312[3175]:= 16#e5ae;
    GB2312[3176]:= 16#b9e0;
    GB2312[3177]:= 16#e5b0;
    GB2312[3178]:= 16#e5b1;
    GB2312[3179]:= 16#bbf0;
    GB2312[3180]:= 16#ece1;
    GB2312[3181]:= 16#c3f0;
    GB2312[3182]:= 16#b5c6;
    GB2312[3183]:= 16#bbd2;
    GB2312[3184]:= 16#c1e9;
    GB2312[3185]:= 16#d4ee;
    GB2312[3186]:= 16#bec4;
    GB2312[3187]:= 16#d7c6;
    GB2312[3188]:= 16#d4d6;
    GB2312[3189]:= 16#b2d3;
    GB2312[3190]:= 16#ecbe;
    GB2312[3191]:= 16#eac1;
    GB2312[3192]:= 16#c2af;
    GB2312[3193]:= 16#b4b6;
    GB2312[3194]:= 16#d1d7;
    GB2312[3195]:= 16#b3b4;
    GB2312[3196]:= 16#c8b2;
    GB2312[3197]:= 16#bfbb;
    GB2312[3198]:= 16#ecc0;
    GB2312[3199]:= 16#d6cb;
    GB2312[3200]:= 16#ecbf;
    GB2312[3201]:= 16#ecc1;
    GB2312[3202]:= 16#ecc5;
    GB2312[3203]:= 16#bee6;
    GB2312[3204]:= 16#ccbf;
    GB2312[3205]:= 16#c5da;
    GB2312[3206]:= 16#bebc;
    GB2312[3207]:= 16#ecc6;
    GB2312[3208]:= 16#b1fe;
    GB2312[3209]:= 16#ecc4;
    GB2312[3210]:= 16#d5a8;
    GB2312[3211]:= 16#b5e3;
    GB2312[3212]:= 16#ecc2;
    GB2312[3213]:= 16#c1b6;
    GB2312[3214]:= 16#b3e3;
    GB2312[3215]:= 16#ecc3;
    GB2312[3216]:= 16#cbb8;
    GB2312[3217]:= 16#c0c3;
    GB2312[3218]:= 16#ccfe;
    GB2312[3219]:= 16#c1d2;
    GB2312[3220]:= 16#ecc8;
    GB2312[3221]:= 16#bae6;
    GB2312[3222]:= 16#c0d3;
    GB2312[3223]:= 16#d6f2;
    GB2312[3224]:= 16#d1cc;
    GB2312[3225]:= 16#bfbe;
    GB2312[3226]:= 16#b7b3;
    GB2312[3227]:= 16#c9d5;
    GB2312[3228]:= 16#ecc7;
    GB2312[3229]:= 16#bbe2;
    GB2312[3230]:= 16#cccc;
    GB2312[3231]:= 16#bdfd;
    GB2312[3232]:= 16#c8c8;
    GB2312[3233]:= 16#cfa9;
    GB2312[3234]:= 16#cde9;
    GB2312[3235]:= 16#c5eb;
    GB2312[3236]:= 16#b7e9;
    GB2312[3237]:= 16#d1c9;
    GB2312[3238]:= 16#bab8;
    GB2312[3239]:= 16#ecc9;
    GB2312[3240]:= 16#ecca;
    GB2312[3241]:= 16#bbc0;
    GB2312[3242]:= 16#eccb;
    GB2312[3243]:= 16#ece2;
    GB2312[3244]:= 16#b1ba;
    GB2312[3245]:= 16#b7d9;
    GB2312[3246]:= 16#bdb9;
    GB2312[3247]:= 16#eccc;
    GB2312[3248]:= 16#d1e6;
    GB2312[3249]:= 16#eccd;
    GB2312[3250]:= 16#c8bb;
    GB2312[3251]:= 16#ecd1;
    GB2312[3252]:= 16#ecd3;
    GB2312[3253]:= 16#bbcd;
    GB2312[3254]:= 16#bce5;
    GB2312[3255]:= 16#eccf;
    GB2312[3256]:= 16#c9b7;
    GB2312[3257]:= 16#c3ba;
    GB2312[3258]:= 16#ece3;
    GB2312[3259]:= 16#d5d5;
    GB2312[3260]:= 16#ecd0;
    GB2312[3261]:= 16#d6f3;
    GB2312[3262]:= 16#ecd2;
    GB2312[3263]:= 16#ecce;
    GB2312[3264]:= 16#ecd4;
    GB2312[3265]:= 16#ecd5;
    GB2312[3266]:= 16#c9bf;
    GB2312[3267]:= 16#cfa8;
    GB2312[3268]:= 16#d0dc;
    GB2312[3269]:= 16#d1ac;
    GB2312[3270]:= 16#c8db;
    GB2312[3271]:= 16#ecd6;
    GB2312[3272]:= 16#cef5;
    GB2312[3273]:= 16#caec;
    GB2312[3274]:= 16#ecda;
    GB2312[3275]:= 16#ecd9;
    GB2312[3276]:= 16#b0be;
    GB2312[3277]:= 16#ecd7;
    GB2312[3278]:= 16#ecd8;
    GB2312[3279]:= 16#ece4;
    GB2312[3280]:= 16#c8bc;
    GB2312[3281]:= 16#c1c7;
    GB2312[3282]:= 16#ecdc;
    GB2312[3283]:= 16#d1e0;
    GB2312[3284]:= 16#ecdb;
    GB2312[3285]:= 16#d4ef;
    GB2312[3286]:= 16#ecdd;
    GB2312[3287]:= 16#dbc6;
    GB2312[3288]:= 16#ecde;
    GB2312[3289]:= 16#b1ac;
    GB2312[3290]:= 16#ecdf;
    GB2312[3291]:= 16#ece0;
    GB2312[3292]:= 16#d7a6;
    GB2312[3293]:= 16#c5c0;
    GB2312[3294]:= 16#ebbc;
    GB2312[3295]:= 16#b0ae;
    GB2312[3296]:= 16#bef4;
    GB2312[3297]:= 16#b8b8;
    GB2312[3298]:= 16#d2af;
    GB2312[3299]:= 16#b0d6;
    GB2312[3300]:= 16#b5f9;
    GB2312[3301]:= 16#d8b3;
    GB2312[3302]:= 16#cbac;
    GB2312[3303]:= 16#e3dd;
    GB2312[3304]:= 16#c6ac;
    GB2312[3305]:= 16#b0e6;
    GB2312[3306]:= 16#c5c6;
    GB2312[3307]:= 16#ebb9;
    GB2312[3308]:= 16#ebba;
    GB2312[3309]:= 16#ebbb;
    GB2312[3310]:= 16#d1c0;
    GB2312[3311]:= 16#c5a3;
    GB2312[3312]:= 16#eaf2;
    GB2312[3313]:= 16#c4b2;
    GB2312[3314]:= 16#c4b5;
    GB2312[3315]:= 16#c0ce;
    GB2312[3316]:= 16#eaf3;
    GB2312[3317]:= 16#c4c1;
    GB2312[3318]:= 16#ceef;
    GB2312[3319]:= 16#eaf0;
    GB2312[3320]:= 16#eaf4;
    GB2312[3321]:= 16#c9fc;
    GB2312[3322]:= 16#c7a3;
    GB2312[3323]:= 16#ccd8;
    GB2312[3324]:= 16#cefe;
    GB2312[3325]:= 16#eaf5;
    GB2312[3326]:= 16#eaf6;
    GB2312[3327]:= 16#cfac;
    GB2312[3328]:= 16#c0e7;
    GB2312[3329]:= 16#eaf7;
    GB2312[3330]:= 16#b6bf;
    GB2312[3331]:= 16#eaf8;
    GB2312[3332]:= 16#eaf9;
    GB2312[3333]:= 16#eafa;
    GB2312[3334]:= 16#eafb;
    GB2312[3335]:= 16#eaf1;
    GB2312[3336]:= 16#c8ae;
    GB2312[3337]:= 16#e1eb;
    GB2312[3338]:= 16#b7b8;
    GB2312[3339]:= 16#e1ec;
    GB2312[3340]:= 16#e1ed;
    GB2312[3341]:= 16#d7b4;
    GB2312[3342]:= 16#e1ee;
    GB2312[3343]:= 16#e1ef;
    GB2312[3344]:= 16#d3cc;
    GB2312[3345]:= 16#e1f1;
    GB2312[3346]:= 16#bff1;
    GB2312[3347]:= 16#e1f0;
    GB2312[3348]:= 16#b5d2;
    GB2312[3349]:= 16#b1b7;
    GB2312[3350]:= 16#e1f3;
    GB2312[3351]:= 16#e1f2;
    GB2312[3352]:= 16#bafc;
    GB2312[3353]:= 16#e1f4;
    GB2312[3354]:= 16#b9b7;
    GB2312[3355]:= 16#bed1;
    GB2312[3356]:= 16#c4fc;
    GB2312[3357]:= 16#badd;
    GB2312[3358]:= 16#bdc6;
    GB2312[3359]:= 16#e1f5;
    GB2312[3360]:= 16#e1f7;
    GB2312[3361]:= 16#b6c0;
    GB2312[3362]:= 16#cfc1;
    GB2312[3363]:= 16#caa8;
    GB2312[3364]:= 16#e1f6;
    GB2312[3365]:= 16#d5f8;
    GB2312[3366]:= 16#d3fc;
    GB2312[3367]:= 16#e1f8;
    GB2312[3368]:= 16#e1fc;
    GB2312[3369]:= 16#e1f9;
    GB2312[3370]:= 16#e1fa;
    GB2312[3371]:= 16#c0ea;
    GB2312[3372]:= 16#e1fe;
    GB2312[3373]:= 16#e2a1;
    GB2312[3374]:= 16#c0c7;
    GB2312[3375]:= 16#e1fb;
    GB2312[3376]:= 16#e1fd;
    GB2312[3377]:= 16#e2a5;
    GB2312[3378]:= 16#c1d4;
    GB2312[3379]:= 16#e2a3;
    GB2312[3380]:= 16#e2a8;
    GB2312[3381]:= 16#b2fe;
    GB2312[3382]:= 16#e2a2;
    GB2312[3383]:= 16#c3cd;
    GB2312[3384]:= 16#b2c2;
    GB2312[3385]:= 16#e2a7;
    GB2312[3386]:= 16#e2a6;
    GB2312[3387]:= 16#e2a4;
    GB2312[3388]:= 16#e2a9;
    GB2312[3389]:= 16#e2ab;
    GB2312[3390]:= 16#d0c9;
    GB2312[3391]:= 16#d6ed;
    GB2312[3392]:= 16#c3a8;
    GB2312[3393]:= 16#e2ac;
    GB2312[3394]:= 16#cfd7;
    GB2312[3395]:= 16#e2ae;
    GB2312[3396]:= 16#baef;
    GB2312[3397]:= 16#e9e0;
    GB2312[3398]:= 16#e2ad;
    GB2312[3399]:= 16#e2aa;
    GB2312[3400]:= 16#bbab;
    GB2312[3401]:= 16#d4b3;
    GB2312[3402]:= 16#e2b0;
    GB2312[3403]:= 16#e2af;
    GB2312[3404]:= 16#e9e1;
    GB2312[3405]:= 16#e2b1;
    GB2312[3406]:= 16#e2b2;
    GB2312[3407]:= 16#e2b3;
    GB2312[3408]:= 16#cca1;
    GB2312[3409]:= 16#e2b4;
    GB2312[3410]:= 16#e2b5;
    GB2312[3411]:= 16#d0fe;
    GB2312[3412]:= 16#c2ca;
    GB2312[3413]:= 16#d3f1;
    GB2312[3414]:= 16#cdf5;
    GB2312[3415]:= 16#e7e0;
    GB2312[3416]:= 16#e7e1;
    GB2312[3417]:= 16#bec1;
    GB2312[3418]:= 16#c2ea;
    GB2312[3419]:= 16#e7e4;
    GB2312[3420]:= 16#e7e3;
    GB2312[3421]:= 16#cde6;
    GB2312[3422]:= 16#c3b5;
    GB2312[3423]:= 16#e7e2;
    GB2312[3424]:= 16#bbb7;
    GB2312[3425]:= 16#cfd6;
    GB2312[3426]:= 16#c1e1;
    GB2312[3427]:= 16#e7e9;
    GB2312[3428]:= 16#e7e8;
    GB2312[3429]:= 16#e7f4;
    GB2312[3430]:= 16#b2a3;
    GB2312[3431]:= 16#e7ea;
    GB2312[3432]:= 16#e7e6;
    GB2312[3433]:= 16#e7ec;
    GB2312[3434]:= 16#e7eb;
    GB2312[3435]:= 16#c9ba;
    GB2312[3436]:= 16#d5e4;
    GB2312[3437]:= 16#e7e5;
    GB2312[3438]:= 16#b7a9;
    GB2312[3439]:= 16#e7e7;
    GB2312[3440]:= 16#e7ee;
    GB2312[3441]:= 16#e7f3;
    GB2312[3442]:= 16#d6e9;
    GB2312[3443]:= 16#e7ed;
    GB2312[3444]:= 16#e7f2;
    GB2312[3445]:= 16#e7f1;
    GB2312[3446]:= 16#b0e0;
    GB2312[3447]:= 16#e7f5;
    GB2312[3448]:= 16#c7f2;
    GB2312[3449]:= 16#c0c5;
    GB2312[3450]:= 16#c0ed;
    GB2312[3451]:= 16#c1f0;
    GB2312[3452]:= 16#e7f0;
    GB2312[3453]:= 16#e7f6;
    GB2312[3454]:= 16#cbf6;
    GB2312[3455]:= 16#e8a2;
    GB2312[3456]:= 16#e8a1;
    GB2312[3457]:= 16#d7c1;
    GB2312[3458]:= 16#e7fa;
    GB2312[3459]:= 16#e7f9;
    GB2312[3460]:= 16#e7fb;
    GB2312[3461]:= 16#e7f7;
    GB2312[3462]:= 16#e7fe;
    GB2312[3463]:= 16#e7fd;
    GB2312[3464]:= 16#e7fc;
    GB2312[3465]:= 16#c1d5;
    GB2312[3466]:= 16#c7d9;
    GB2312[3467]:= 16#c5fd;
    GB2312[3468]:= 16#c5c3;
    GB2312[3469]:= 16#c7ed;
    GB2312[3470]:= 16#e8a3;
    GB2312[3471]:= 16#e8a6;
    GB2312[3472]:= 16#e8a5;
    GB2312[3473]:= 16#e8a7;
    GB2312[3474]:= 16#baf7;
    GB2312[3475]:= 16#e7f8;
    GB2312[3476]:= 16#e8a4;
    GB2312[3477]:= 16#c8f0;
    GB2312[3478]:= 16#c9aa;
    GB2312[3479]:= 16#e8a9;
    GB2312[3480]:= 16#b9e5;
    GB2312[3481]:= 16#d1fe;
    GB2312[3482]:= 16#e8a8;
    GB2312[3483]:= 16#e8aa;
    GB2312[3484]:= 16#e8ad;
    GB2312[3485]:= 16#e8ae;
    GB2312[3486]:= 16#c1a7;
    GB2312[3487]:= 16#e8af;
    GB2312[3488]:= 16#e8b0;
    GB2312[3489]:= 16#e8ac;
    GB2312[3490]:= 16#e8b4;
    GB2312[3491]:= 16#e8ab;
    GB2312[3492]:= 16#e8b1;
    GB2312[3493]:= 16#e8b5;
    GB2312[3494]:= 16#e8b2;
    GB2312[3495]:= 16#e8b3;
    GB2312[3496]:= 16#e8b7;
    GB2312[3497]:= 16#e8b6;
    GB2312[3498]:= 16#b9cf;
    GB2312[3499]:= 16#f0ac;
    GB2312[3500]:= 16#f0ad;
    GB2312[3501]:= 16#c6b0;
    GB2312[3502]:= 16#b0ea;
    GB2312[3503]:= 16#c8bf;
    GB2312[3504]:= 16#cddf;
    GB2312[3505]:= 16#cecd;
    GB2312[3506]:= 16#eab1;
    GB2312[3507]:= 16#eab2;
    GB2312[3508]:= 16#c6bf;
    GB2312[3509]:= 16#b4c9;
    GB2312[3510]:= 16#eab3;
    GB2312[3511]:= 16#d5e7;
    GB2312[3512]:= 16#ddf9;
    GB2312[3513]:= 16#eab4;
    GB2312[3514]:= 16#eab5;
    GB2312[3515]:= 16#eab6;
    GB2312[3516]:= 16#b8ca;
    GB2312[3517]:= 16#dfb0;
    GB2312[3518]:= 16#c9f5;
    GB2312[3519]:= 16#ccf0;
    GB2312[3520]:= 16#c9fa;
    GB2312[3521]:= 16#c9fb;
    GB2312[3522]:= 16#d3c3;
    GB2312[3523]:= 16#cba6;
    GB2312[3524]:= 16#b8a6;
    GB2312[3525]:= 16#f0ae;
    GB2312[3526]:= 16#b1c2;
    GB2312[3527]:= 16#e5b8;
    GB2312[3528]:= 16#ccef;
    GB2312[3529]:= 16#d3c9;
    GB2312[3530]:= 16#bcd7;
    GB2312[3531]:= 16#c9ea;
    GB2312[3532]:= 16#b5e7;
    GB2312[3533]:= 16#c4d0;
    GB2312[3534]:= 16#b5e9;
    GB2312[3535]:= 16#eeae;
    GB2312[3536]:= 16#bbad;
    GB2312[3537]:= 16#e7de;
    GB2312[3538]:= 16#eeaf;
    GB2312[3539]:= 16#b3a9;
    GB2312[3540]:= 16#eeb2;
    GB2312[3541]:= 16#eeb1;
    GB2312[3542]:= 16#bde7;
    GB2312[3543]:= 16#eeb0;
    GB2312[3544]:= 16#ceb7;
    GB2312[3545]:= 16#c5cf;
    GB2312[3546]:= 16#c1f4;
    GB2312[3547]:= 16#dbce;
    GB2312[3548]:= 16#eeb3;
    GB2312[3549]:= 16#d0f3;
    GB2312[3550]:= 16#c2d4;
    GB2312[3551]:= 16#c6e8;
    GB2312[3552]:= 16#b7ac;
    GB2312[3553]:= 16#eeb4;
    GB2312[3554]:= 16#b3eb;
    GB2312[3555]:= 16#bbfb;
    GB2312[3556]:= 16#eeb5;
    GB2312[3557]:= 16#e7dc;
    GB2312[3558]:= 16#eeb6;
    GB2312[3559]:= 16#bdae;
    GB2312[3560]:= 16#f1e2;
    GB2312[3561]:= 16#cae8;
    GB2312[3562]:= 16#d2c9;
    GB2312[3563]:= 16#f0da;
    GB2312[3564]:= 16#f0db;
    GB2312[3565]:= 16#f0dc;
    GB2312[3566]:= 16#c1c6;
    GB2312[3567]:= 16#b8ed;
    GB2312[3568]:= 16#bece;
    GB2312[3569]:= 16#f0de;
    GB2312[3570]:= 16#c5b1;
    GB2312[3571]:= 16#f0dd;
    GB2312[3572]:= 16#d1f1;
    GB2312[3573]:= 16#f0e0;
    GB2312[3574]:= 16#b0cc;
    GB2312[3575]:= 16#bdea;
    GB2312[3576]:= 16#d2df;
    GB2312[3577]:= 16#f0df;
    GB2312[3578]:= 16#b4af;
    GB2312[3579]:= 16#b7e8;
    GB2312[3580]:= 16#f0e6;
    GB2312[3581]:= 16#f0e5;
    GB2312[3582]:= 16#c6a3;
    GB2312[3583]:= 16#f0e1;
    GB2312[3584]:= 16#f0e2;
    GB2312[3585]:= 16#b4c3;
    GB2312[3586]:= 16#f0e3;
    GB2312[3587]:= 16#d5ee;
    GB2312[3588]:= 16#ccdb;
    GB2312[3589]:= 16#bed2;
    GB2312[3590]:= 16#bcb2;
    GB2312[3591]:= 16#f0e8;
    GB2312[3592]:= 16#f0e7;
    GB2312[3593]:= 16#f0e4;
    GB2312[3594]:= 16#b2a1;
    GB2312[3595]:= 16#d6a2;
    GB2312[3596]:= 16#d3b8;
    GB2312[3597]:= 16#beb7;
    GB2312[3598]:= 16#c8ac;
    GB2312[3599]:= 16#f0ea;
    GB2312[3600]:= 16#d1f7;
    GB2312[3601]:= 16#d6cc;
    GB2312[3602]:= 16#badb;
    GB2312[3603]:= 16#f0e9;
    GB2312[3604]:= 16#b6bb;
    GB2312[3605]:= 16#cdb4;
    GB2312[3606]:= 16#c6a6;
    GB2312[3607]:= 16#c1a1;
    GB2312[3608]:= 16#f0eb;
    GB2312[3609]:= 16#f0ee;
    GB2312[3610]:= 16#f0ed;
    GB2312[3611]:= 16#f0f0;
    GB2312[3612]:= 16#f0ec;
    GB2312[3613]:= 16#bbbe;
    GB2312[3614]:= 16#f0ef;
    GB2312[3615]:= 16#ccb5;
    GB2312[3616]:= 16#f0f2;
    GB2312[3617]:= 16#b3d5;
    GB2312[3618]:= 16#b1d4;
    GB2312[3619]:= 16#f0f3;
    GB2312[3620]:= 16#f0f4;
    GB2312[3621]:= 16#f0f6;
    GB2312[3622]:= 16#b4e1;
    GB2312[3623]:= 16#f0f1;
    GB2312[3624]:= 16#f0f7;
    GB2312[3625]:= 16#f0fa;
    GB2312[3626]:= 16#f0f8;
    GB2312[3627]:= 16#f0f5;
    GB2312[3628]:= 16#f0fd;
    GB2312[3629]:= 16#f0f9;
    GB2312[3630]:= 16#f0fc;
    GB2312[3631]:= 16#f0fe;
    GB2312[3632]:= 16#f1a1;
    GB2312[3633]:= 16#cec1;
    GB2312[3634]:= 16#f1a4;
    GB2312[3635]:= 16#f1a3;
    GB2312[3636]:= 16#c1f6;
    GB2312[3637]:= 16#f0fb;
    GB2312[3638]:= 16#cadd;
    GB2312[3639]:= 16#b4f1;
    GB2312[3640]:= 16#b1f1;
    GB2312[3641]:= 16#ccb1;
    GB2312[3642]:= 16#f1a6;
    GB2312[3643]:= 16#f1a7;
    GB2312[3644]:= 16#f1ac;
    GB2312[3645]:= 16#d5ce;
    GB2312[3646]:= 16#f1a9;
    GB2312[3647]:= 16#c8b3;
    GB2312[3648]:= 16#f1a2;
    GB2312[3649]:= 16#f1ab;
    GB2312[3650]:= 16#f1a8;
    GB2312[3651]:= 16#f1a5;
    GB2312[3652]:= 16#f1aa;
    GB2312[3653]:= 16#b0a9;
    GB2312[3654]:= 16#f1ad;
    GB2312[3655]:= 16#f1af;
    GB2312[3656]:= 16#f1b1;
    GB2312[3657]:= 16#f1b0;
    GB2312[3658]:= 16#f1ae;
    GB2312[3659]:= 16#d1a2;
    GB2312[3660]:= 16#f1b2;
    GB2312[3661]:= 16#f1b3;
    GB2312[3662]:= 16#b9ef;
    GB2312[3663]:= 16#b5c7;
    GB2312[3664]:= 16#b0d7;
    GB2312[3665]:= 16#b0d9;
    GB2312[3666]:= 16#d4ed;
    GB2312[3667]:= 16#b5c4;
    GB2312[3668]:= 16#bdd4;
    GB2312[3669]:= 16#bbca;
    GB2312[3670]:= 16#f0a7;
    GB2312[3671]:= 16#b8de;
    GB2312[3672]:= 16#f0a8;
    GB2312[3673]:= 16#b0a8;
    GB2312[3674]:= 16#f0a9;
    GB2312[3675]:= 16#cdee;
    GB2312[3676]:= 16#f0aa;
    GB2312[3677]:= 16#f0ab;
    GB2312[3678]:= 16#c6a4;
    GB2312[3679]:= 16#d6e5;
    GB2312[3680]:= 16#f1e4;
    GB2312[3681]:= 16#f1e5;
    GB2312[3682]:= 16#c3f3;
    GB2312[3683]:= 16#d3db;
    GB2312[3684]:= 16#d6d1;
    GB2312[3685]:= 16#c5e8;
    GB2312[3686]:= 16#d3af;
    GB2312[3687]:= 16#d2e6;
    GB2312[3688]:= 16#eec1;
    GB2312[3689]:= 16#b0bb;
    GB2312[3690]:= 16#d5b5;
    GB2312[3691]:= 16#d1ce;
    GB2312[3692]:= 16#bce0;
    GB2312[3693]:= 16#bad0;
    GB2312[3694]:= 16#bff8;
    GB2312[3695]:= 16#b8c7;
    GB2312[3696]:= 16#b5c1;
    GB2312[3697]:= 16#c5cc;
    GB2312[3698]:= 16#caa2;
    GB2312[3699]:= 16#c3cb;
    GB2312[3700]:= 16#eec2;
    GB2312[3701]:= 16#c4bf;
    GB2312[3702]:= 16#b6a2;
    GB2312[3703]:= 16#edec;
    GB2312[3704]:= 16#c3a4;
    GB2312[3705]:= 16#d6b1;
    GB2312[3706]:= 16#cfe0;
    GB2312[3707]:= 16#edef;
    GB2312[3708]:= 16#c5ce;
    GB2312[3709]:= 16#b6dc;
    GB2312[3710]:= 16#caa1;
    GB2312[3711]:= 16#eded;
    GB2312[3712]:= 16#edf0;
    GB2312[3713]:= 16#edf1;
    GB2312[3714]:= 16#c3bc;
    GB2312[3715]:= 16#bfb4;
    GB2312[3716]:= 16#edee;
    GB2312[3717]:= 16#edf4;
    GB2312[3718]:= 16#edf2;
    GB2312[3719]:= 16#d5e6;
    GB2312[3720]:= 16#c3df;
    GB2312[3721]:= 16#edf3;
    GB2312[3722]:= 16#edf6;
    GB2312[3723]:= 16#d5a3;
    GB2312[3724]:= 16#d1a3;
    GB2312[3725]:= 16#edf5;
    GB2312[3726]:= 16#c3d0;
    GB2312[3727]:= 16#edf7;
    GB2312[3728]:= 16#bff4;
    GB2312[3729]:= 16#beec;
    GB2312[3730]:= 16#edf8;
    GB2312[3731]:= 16#ccf7;
    GB2312[3732]:= 16#d1db;
    GB2312[3733]:= 16#d7c5;
    GB2312[3734]:= 16#d5f6;
    GB2312[3735]:= 16#edfc;
    GB2312[3736]:= 16#edfb;
    GB2312[3737]:= 16#edf9;
    GB2312[3738]:= 16#edfa;
    GB2312[3739]:= 16#edfd;
    GB2312[3740]:= 16#bea6;
    GB2312[3741]:= 16#cbaf;
    GB2312[3742]:= 16#eea1;
    GB2312[3743]:= 16#b6bd;
    GB2312[3744]:= 16#eea2;
    GB2312[3745]:= 16#c4c0;
    GB2312[3746]:= 16#edfe;
    GB2312[3747]:= 16#bdde;
    GB2312[3748]:= 16#b2c7;
    GB2312[3749]:= 16#b6c3;
    GB2312[3750]:= 16#eea5;
    GB2312[3751]:= 16#d8ba;
    GB2312[3752]:= 16#eea3;
    GB2312[3753]:= 16#eea6;
    GB2312[3754]:= 16#c3e9;
    GB2312[3755]:= 16#b3f2;
    GB2312[3756]:= 16#eea7;
    GB2312[3757]:= 16#eea4;
    GB2312[3758]:= 16#cfb9;
    GB2312[3759]:= 16#eea8;
    GB2312[3760]:= 16#c2f7;
    GB2312[3761]:= 16#eea9;
    GB2312[3762]:= 16#eeaa;
    GB2312[3763]:= 16#deab;
    GB2312[3764]:= 16#c6b3;
    GB2312[3765]:= 16#c7c6;
    GB2312[3766]:= 16#d6f5;
    GB2312[3767]:= 16#b5c9;
    GB2312[3768]:= 16#cbb2;
    GB2312[3769]:= 16#eeab;
    GB2312[3770]:= 16#cdab;
    GB2312[3771]:= 16#eeac;
    GB2312[3772]:= 16#d5b0;
    GB2312[3773]:= 16#eead;
    GB2312[3774]:= 16#f6c4;
    GB2312[3775]:= 16#dbc7;
    GB2312[3776]:= 16#b4a3;
    GB2312[3777]:= 16#c3ac;
    GB2312[3778]:= 16#f1e6;
    GB2312[3779]:= 16#cab8;
    GB2312[3780]:= 16#d2d3;
    GB2312[3781]:= 16#d6aa;
    GB2312[3782]:= 16#eff2;
    GB2312[3783]:= 16#bed8;
    GB2312[3784]:= 16#bdc3;
    GB2312[3785]:= 16#eff3;
    GB2312[3786]:= 16#b6cc;
    GB2312[3787]:= 16#b0ab;
    GB2312[3788]:= 16#caaf;
    GB2312[3789]:= 16#edb6;
    GB2312[3790]:= 16#edb7;
    GB2312[3791]:= 16#cef9;
    GB2312[3792]:= 16#b7af;
    GB2312[3793]:= 16#bff3;
    GB2312[3794]:= 16#edb8;
    GB2312[3795]:= 16#c2eb;
    GB2312[3796]:= 16#c9b0;
    GB2312[3797]:= 16#edb9;
    GB2312[3798]:= 16#c6f6;
    GB2312[3799]:= 16#bfb3;
    GB2312[3800]:= 16#edbc;
    GB2312[3801]:= 16#c5f8;
    GB2312[3802]:= 16#d1d0;
    GB2312[3803]:= 16#d7a9;
    GB2312[3804]:= 16#edba;
    GB2312[3805]:= 16#edbb;
    GB2312[3806]:= 16#d1e2;
    GB2312[3807]:= 16#edbf;
    GB2312[3808]:= 16#edc0;
    GB2312[3809]:= 16#edc4;
    GB2312[3810]:= 16#edc8;
    GB2312[3811]:= 16#edc6;
    GB2312[3812]:= 16#edce;
    GB2312[3813]:= 16#d5e8;
    GB2312[3814]:= 16#edc9;
    GB2312[3815]:= 16#edc7;
    GB2312[3816]:= 16#edbe;
    GB2312[3817]:= 16#c5e9;
    GB2312[3818]:= 16#c6c6;
    GB2312[3819]:= 16#c9e9;
    GB2312[3820]:= 16#d4d2;
    GB2312[3821]:= 16#edc1;
    GB2312[3822]:= 16#edc2;
    GB2312[3823]:= 16#edc3;
    GB2312[3824]:= 16#edc5;
    GB2312[3825]:= 16#c0f9;
    GB2312[3826]:= 16#b4a1;
    GB2312[3827]:= 16#b9e8;
    GB2312[3828]:= 16#edd0;
    GB2312[3829]:= 16#edd1;
    GB2312[3830]:= 16#edca;
    GB2312[3831]:= 16#edcf;
    GB2312[3832]:= 16#cef8;
    GB2312[3833]:= 16#cbb6;
    GB2312[3834]:= 16#edcc;
    GB2312[3835]:= 16#edcd;
    GB2312[3836]:= 16#cff5;
    GB2312[3837]:= 16#edd2;
    GB2312[3838]:= 16#c1f2;
    GB2312[3839]:= 16#d3b2;
    GB2312[3840]:= 16#edcb;
    GB2312[3841]:= 16#c8b7;
    GB2312[3842]:= 16#bcef;
    GB2312[3843]:= 16#c5f0;
    GB2312[3844]:= 16#edd6;
    GB2312[3845]:= 16#b5ef;
    GB2312[3846]:= 16#c2b5;
    GB2312[3847]:= 16#b0ad;
    GB2312[3848]:= 16#cbe9;
    GB2312[3849]:= 16#b1ae;
    GB2312[3850]:= 16#edd4;
    GB2312[3851]:= 16#cdeb;
    GB2312[3852]:= 16#b5e2;
    GB2312[3853]:= 16#edd5;
    GB2312[3854]:= 16#edd3;
    GB2312[3855]:= 16#edd7;
    GB2312[3856]:= 16#b5fa;
    GB2312[3857]:= 16#edd8;
    GB2312[3858]:= 16#edd9;
    GB2312[3859]:= 16#eddc;
    GB2312[3860]:= 16#b1cc;
    GB2312[3861]:= 16#c5f6;
    GB2312[3862]:= 16#bcee;
    GB2312[3863]:= 16#edda;
    GB2312[3864]:= 16#ccbc;
    GB2312[3865]:= 16#b2ea;
    GB2312[3866]:= 16#eddb;
    GB2312[3867]:= 16#c4eb;
    GB2312[3868]:= 16#b4c5;
    GB2312[3869]:= 16#b0f5;
    GB2312[3870]:= 16#eddf;
    GB2312[3871]:= 16#c0da;
    GB2312[3872]:= 16#b4e8;
    GB2312[3873]:= 16#c5cd;
    GB2312[3874]:= 16#eddd;
    GB2312[3875]:= 16#bfc4;
    GB2312[3876]:= 16#edde;
    GB2312[3877]:= 16#c4a5;
    GB2312[3878]:= 16#ede0;
    GB2312[3879]:= 16#ede1;
    GB2312[3880]:= 16#ede3;
    GB2312[3881]:= 16#c1d7;
    GB2312[3882]:= 16#bbc7;
    GB2312[3883]:= 16#bdb8;
    GB2312[3884]:= 16#ede2;
    GB2312[3885]:= 16#ede4;
    GB2312[3886]:= 16#ede6;
    GB2312[3887]:= 16#ede5;
    GB2312[3888]:= 16#ede7;
    GB2312[3889]:= 16#cabe;
    GB2312[3890]:= 16#ecea;
    GB2312[3891]:= 16#c0f1;
    GB2312[3892]:= 16#c9e7;
    GB2312[3893]:= 16#eceb;
    GB2312[3894]:= 16#c6ee;
    GB2312[3895]:= 16#ecec;
    GB2312[3896]:= 16#c6ed;
    GB2312[3897]:= 16#eced;
    GB2312[3898]:= 16#ecf0;
    GB2312[3899]:= 16#d7e6;
    GB2312[3900]:= 16#ecf3;
    GB2312[3901]:= 16#ecf1;
    GB2312[3902]:= 16#ecee;
    GB2312[3903]:= 16#ecef;
    GB2312[3904]:= 16#d7a3;
    GB2312[3905]:= 16#c9f1;
    GB2312[3906]:= 16#cbee;
    GB2312[3907]:= 16#ecf4;
    GB2312[3908]:= 16#ecf2;
    GB2312[3909]:= 16#cfe9;
    GB2312[3910]:= 16#ecf6;
    GB2312[3911]:= 16#c6b1;
    GB2312[3912]:= 16#bcc0;
    GB2312[3913]:= 16#ecf5;
    GB2312[3914]:= 16#b5bb;
    GB2312[3915]:= 16#bbf6;
    GB2312[3916]:= 16#ecf7;
    GB2312[3917]:= 16#d9f7;
    GB2312[3918]:= 16#bdfb;
    GB2312[3919]:= 16#c2bb;
    GB2312[3920]:= 16#ecf8;
    GB2312[3921]:= 16#ecf9;
    GB2312[3922]:= 16#b8a3;
    GB2312[3923]:= 16#ecfa;
    GB2312[3924]:= 16#ecfb;
    GB2312[3925]:= 16#ecfc;
    GB2312[3926]:= 16#d3ed;
    GB2312[3927]:= 16#d8ae;
    GB2312[3928]:= 16#c0eb;
    GB2312[3929]:= 16#c7dd;
    GB2312[3930]:= 16#bacc;
    GB2312[3931]:= 16#d0e3;
    GB2312[3932]:= 16#cbbd;
    GB2312[3933]:= 16#cdba;
    GB2312[3934]:= 16#b8d1;
    GB2312[3935]:= 16#b1fc;
    GB2312[3936]:= 16#c7ef;
    GB2312[3937]:= 16#d6d6;
    GB2312[3938]:= 16#bfc6;
    GB2312[3939]:= 16#c3eb;
    GB2312[3940]:= 16#eff5;
    GB2312[3941]:= 16#c3d8;
    GB2312[3942]:= 16#d7e2;
    GB2312[3943]:= 16#eff7;
    GB2312[3944]:= 16#b3d3;
    GB2312[3945]:= 16#c7d8;
    GB2312[3946]:= 16#d1ed;
    GB2312[3947]:= 16#d6c8;
    GB2312[3948]:= 16#eff8;
    GB2312[3949]:= 16#eff6;
    GB2312[3950]:= 16#bbfd;
    GB2312[3951]:= 16#b3c6;
    GB2312[3952]:= 16#bdd5;
    GB2312[3953]:= 16#d2c6;
    GB2312[3954]:= 16#bbe0;
    GB2312[3955]:= 16#cfa1;
    GB2312[3956]:= 16#effc;
    GB2312[3957]:= 16#effb;
    GB2312[3958]:= 16#eff9;
    GB2312[3959]:= 16#b3cc;
    GB2312[3960]:= 16#c9d4;
    GB2312[3961]:= 16#cbb0;
    GB2312[3962]:= 16#effe;
    GB2312[3963]:= 16#b0de;
    GB2312[3964]:= 16#d6c9;
    GB2312[3965]:= 16#effd;
    GB2312[3966]:= 16#b3ed;
    GB2312[3967]:= 16#f6d5;
    GB2312[3968]:= 16#cec8;
    GB2312[3969]:= 16#f0a2;
    GB2312[3970]:= 16#f0a1;
    GB2312[3971]:= 16#b5be;
    GB2312[3972]:= 16#bcda;
    GB2312[3973]:= 16#bbfc;
    GB2312[3974]:= 16#b8e5;
    GB2312[3975]:= 16#c4c2;
    GB2312[3976]:= 16#f0a3;
    GB2312[3977]:= 16#cbeb;
    GB2312[3978]:= 16#f0a6;
    GB2312[3979]:= 16#d1a8;
    GB2312[3980]:= 16#bebf;
    GB2312[3981]:= 16#c7ee;
